LIN {X 0.072,Y -139.487,Z 751.117,A 0.000,B 0.000,C 90.000,E1 200.972} C_DIS
LIN {X 0.061,Y -138.989,Z 751.101,A 0.000,B 0.000,C 90.000,E1 198.181} C_DIS
LIN {X 0.022,Y -138.335,Z 751.054,A 0.000,B 0.000,C 90.000,E1 189.792} C_DIS
LIN {X 0.046,Y -139.420,Z 751.008,A 0.000,B 0.000,C 90.000,E1 181.375} C_DIS
LIN {X -0.041,Y -141.340,Z 750.972,A 0.000,B 0.000,C 90.000,E1 174.894} C_DIS
LIN {X 0.078,Y -142.696,Z 750.956,A 0.000,B 0.000,C 90.000,E1 172.064} C_DIS
LIN {X 0.038,Y -145.062,Z 750.930,A 0.000,B 0.000,C 90.000,E1 167.465} C_DIS
LIN {X 0.034,Y -147.687,Z 750.910,A 0.000,B 0.000,C 90.000,E1 163.795} C_DIS
LIN {X -0.074,Y -150.334,Z 750.890,A 0.000,B 0.000,C 90.000,E1 160.188} C_DIS
LIN {X -0.003,Y -153.753,Z 750.870,A 0.000,B 0.000,C 90.000,E1 156.538} C_DIS
LIN {X -0.012,Y -157.166,Z 750.850,A 0.000,B 0.000,C 90.000,E1 152.948} C_DIS
LIN {X -0.078,Y -161.320,Z 750.830,A 0.000,B 0.000,C 90.000,E1 149.410} C_DIS
LIN {X 0.075,Y -164.434,Z 750.815,A 0.000,B 0.000,C 90.000,E1 146.707} C_DIS
LIN {X 0.070,Y -169.120,Z 750.796,A 0.000,B 0.000,C 90.000,E1 143.210} C_DIS
LIN {X 0.018,Y -171.673,Z 750.786,A 0.000,B 0.000,C 90.000,E1 141.492} C_DIS
LIN {X -0.070,Y -176.641,Z 750.767,A 0.000,B 0.000,C 90.000,E1 138.081} C_DIS
LIN {X 0.057,Y -180.939,Z 750.753,A 0.000,B 0.000,C 90.000,E1 135.486} C_DIS
LIN {X 0.045,Y -186.359,Z 750.734,A 0.000,B 0.000,C 90.000,E1 132.123} C_DIS
LIN {X 0.004,Y -191.446,Z 750.719,A 0.000,B 0.000,C 90.000,E1 129.358} C_DIS
LIN {X 0.019,Y -192.042,Z 750.717,A 0.000,B 0.000,C 90.000,E1 128.991} C_DIS
LIN {X -0.007,Y -291.468,Z 750.717,A 0.000,B 0.000,C 90.000,E1 128.991} C_DIS
LIN {X -0.087,Y -296.497,Z 750.716,A 0.000,B 0.000,C 90.000,E1 128.830} C_DIS
LIN {X 0.018,Y -299.370,Z 750.714,A 0.000,B 0.000,C 90.000,E1 128.588} C_DIS
LIN {X -0.036,Y -303.124,Z 750.712,A 0.000,B 0.000,C 90.000,E1 128.141} C_DIS
LIN {X -0.019,Y -304.997,Z 750.710,A 0.000,B 0.000,C 90.000,E1 127.810} C_DIS
LIN {X 0.187,Y -306.459,Z 750.708,A 0.000,B 0.000,C 90.000,E1 127.443} C_DIS
LIN {X 0.173,Y -308.546,Z 750.705,A 0.000,B 0.000,C 90.000,E1 126.790} C_DIS
LIN {X -0.011,Y -318.461,Z 750.687,A 0.000,B 0.000,C 90.000,E1 123.579} C_DIS
LIN {X -0.052,Y -328.690,Z 750.671,A 0.000,B 0.000,C 90.000,E1 120.718} C_DIS
LIN {X -0.027,Y -340.261,Z 750.655,A 0.000,B 0.000,C 90.000,E1 117.897} C_DIS
LIN {X -0.136,Y -353.272,Z 750.640,A 0.000,B 0.000,C 90.000,E1 115.155} C_DIS
LIN {X 0.090,Y -366.144,Z 750.626,A 0.000,B 0.000,C 90.000,E1 112.717} C_DIS
LIN {X 0.031,Y -380.339,Z 750.613,A 0.000,B 0.000,C 90.000,E1 110.375} C_DIS
LIN {X 0.187,Y -395.960,Z 750.600,A 0.000,B 0.000,C 90.000,E1 108.055} C_DIS
LIN {X -0.022,Y -413.120,Z 750.588,A 0.000,B 0.000,C 90.000,E1 105.843} C_DIS
LIN {X 0.073,Y -431.944,Z 750.576,A 0.000,B 0.000,C 90.000,E1 103.647} C_DIS
LIN {X 0.019,Y -451.968,Z 750.564,A 0.000,B 0.000,C 90.000,E1 101.591} C_DIS
LIN {X 0.143,Y -467.357,Z 750.556,A 0.000,B 0.000,C 90.000,E1 100.141} C_DIS
LIN {X 0.178,Y -469.582,Z 750.555,A 0.000,B 0.000,C 90.000,E1 99.905} C_DIS
LIN {X 0.030,Y -471.399,Z 750.554,A 0.000,B 0.000,C 90.000,E1 99.670} C_DIS
LIN {X -0.120,Y -472.764,Z 750.552,A 0.000,B 0.000,C 90.000,E1 99.434} C_DIS
LIN {X -0.015,Y -474.484,Z 750.549,A 0.000,B 0.000,C 90.000,E1 98.916} C_DIS
LIN {X 0.102,Y -475.129,Z 750.547,A 0.000,B 0.000,C 90.000,E1 98.398} C_DIS
LIN {X -0.240,Y -474.807,Z 750.544,A 0.000,B 0.000,C 90.000,E1 97.936} C_DIS
LIN {X -0.045,Y -473.473,Z 750.541,A 0.000,B 0.000,C 90.000,E1 97.409} C_DIS
LIN {X -0.245,Y -472.363,Z 750.540,A 0.000,B 0.000,C 90.000,E1 97.182} C_DIS
LIN {X 0.198,Y -467.575,Z 750.536,A 0.000,B 0.000,C 90.000,E1 96.372} C_DIS
LIN {X -0.019,Y -451.599,Z 750.521,A 0.000,B 0.000,C 90.000,E1 93.841} C_DIS
LIN {X -0.186,Y -439.674,Z 750.510,A 0.000,B 0.000,C 90.000,E1 91.776} C_DIS
LIN {X 0.206,Y -432.077,Z 750.502,A 0.000,B 0.000,C 90.000,E1 90.401} C_DIS
LIN {X -0.117,Y -421.060,Z 750.492,A 0.000,B 0.000,C 90.000,E1 88.568} C_DIS
LIN {X 0.197,Y -410.004,Z 750.481,A 0.000,B 0.000,C 90.000,E1 86.617} C_DIS
LIN {X -0.167,Y -400.346,Z 750.472,A 0.000,B 0.000,C 90.000,E1 85.008} C_DIS
LIN {X 0.186,Y -387.551,Z 750.460,A 0.000,B 0.000,C 90.000,E1 82.704} C_DIS
LIN {X -0.043,Y -373.543,Z 750.445,A 0.000,B 0.000,C 90.000,E1 80.151} C_DIS
LIN {X -0.102,Y -361.605,Z 750.432,A 0.000,B 0.000,C 90.000,E1 77.813} C_DIS
LIN {X -0.027,Y -350.077,Z 750.419,A 0.000,B 0.000,C 90.000,E1 75.408} C_DIS
LIN {X 0.024,Y -338.783,Z 750.405,A 0.000,B 0.000,C 90.000,E1 72.960} C_DIS
LIN {X -0.133,Y -326.444,Z 750.390,A 0.000,B 0.000,C 90.000,E1 70.188} C_DIS
LIN {X 0.059,Y -313.531,Z 750.372,A 0.000,B 0.000,C 90.000,E1 66.975} C_DIS
LIN {X 0.121,Y -300.774,Z 750.352,A 0.000,B 0.000,C 90.000,E1 63.384} C_DIS
LIN {X 0.056,Y -290.366,Z 750.334,A 0.000,B 0.000,C 90.000,E1 60.078} C_DIS
LIN {X 0.009,Y -280.599,Z 750.315,A 0.000,B 0.000,C 90.000,E1 56.707} C_DIS
LIN {X -0.136,Y -273.069,Z 750.300,A 0.000,B 0.000,C 90.000,E1 53.989} C_DIS
LIN {X 0.017,Y -265.664,Z 750.284,A 0.000,B 0.000,C 90.000,E1 51.170} C_DIS
LIN {X 0.004,Y -259.989,Z 750.273,A 0.000,B 0.000,C 90.000,E1 49.057} C_DIS
LIN {X 0.056,Y -254.309,Z 750.261,A 0.000,B 0.000,C 90.000,E1 46.905} C_DIS
LIN {X -0.012,Y -248.565,Z 750.249,A 0.000,B 0.000,C 90.000,E1 44.757} C_DIS
LIN {X 0.160,Y -242.844,Z 750.236,A 0.000,B 0.000,C 90.000,E1 42.528} C_DIS
LIN {X -0.147,Y -235.195,Z 750.220,A 0.000,B 0.000,C 90.000,E1 39.644} C_DIS
LIN {X 0.087,Y -227.868,Z 750.203,A 0.000,B 0.000,C 90.000,E1 36.583} C_DIS
LIN {X -0.051,Y -219.365,Z 750.182,A 0.000,B 0.000,C 90.000,E1 32.801} C_DIS
LIN {X 0.065,Y -213.121,Z 750.165,A 0.000,B 0.000,C 90.000,E1 29.667} C_DIS
LIN {X 0.003,Y -207.678,Z 750.147,A 0.000,B 0.000,C 90.000,E1 26.539} C_DIS
LIN {X -0.103,Y -201.882,Z 750.125,A 0.000,B 0.000,C 90.000,E1 22.589} C_DIS
LIN {X -0.047,Y -197.159,Z 750.103,A 0.000,B 0.000,C 90.000,E1 18.544} C_DIS
LIN {X -0.070,Y -193.575,Z 750.080,A 0.000,B 0.000,C 90.000,E1 14.481} C_DIS
LIN {X 0.078,Y -190.269,Z 750.048,A 0.000,B 0.000,C 90.000,E1 8.690} C_DIS
LIN {X -0.039,Y -191.325,Z 749.961,A 0.000,B 0.000,C 90.000,E1 352.932} C_DIS
LIN {X -0.014,Y -194.658,Z 749.933,A 0.000,B 0.000,C 90.000,E1 347.993} C_DIS
LIN {X -0.037,Y -198.529,Z 749.911,A 0.000,B 0.000,C 90.000,E1 343.921} C_DIS
LIN {X -0.043,Y -203.397,Z 749.888,A 0.000,B 0.000,C 90.000,E1 339.880} C_DIS
LIN {X 0.004,Y -209.211,Z 749.866,A 0.000,B 0.000,C 90.000,E1 335.869} C_DIS
LIN {X 0.101,Y -215.898,Z 749.844,A 0.000,B 0.000,C 90.000,E1 331.897} C_DIS
LIN {X -0.033,Y -223.327,Z 749.822,A 0.000,B 0.000,C 90.000,E1 328.043} C_DIS
LIN {X 0.046,Y -231.309,Z 749.801,A 0.000,B 0.000,C 90.000,E1 324.196} C_DIS
LIN {X 0.029,Y -239.935,Z 749.780,A 0.000,B 0.000,C 90.000,E1 320.436} C_DIS
LIN {X 0.035,Y -247.397,Z 749.764,A 0.000,B 0.000,C 90.000,E1 317.472} C_DIS
LIN {X 0.063,Y -256.588,Z 749.746,A 0.000,B 0.000,C 90.000,E1 314.190} C_DIS
LIN {X 0.076,Y -267.646,Z 749.726,A 0.000,B 0.000,C 90.000,E1 310.620} C_DIS
LIN {X -0.048,Y -279.888,Z 749.706,A 0.000,B 0.000,C 90.000,E1 307.156} C_DIS
LIN {X 0.017,Y -291.945,Z 749.689,A 0.000,B 0.000,C 90.000,E1 304.072} C_DIS
LIN {X 0.091,Y -304.024,Z 749.674,A 0.000,B 0.000,C 90.000,E1 301.386} C_DIS
LIN {X -0.036,Y -320.894,Z 749.656,A 0.000,B 0.000,C 90.000,E1 298.153} C_DIS
LIN {X 0.011,Y -333.660,Z 749.644,A 0.000,B 0.000,C 90.000,E1 295.924} C_DIS
LIN {X 0.062,Y -351.261,Z 749.629,A 0.000,B 0.000,C 90.000,E1 293.131} C_DIS
LIN {X 0.151,Y -372.539,Z 749.612,A 0.000,B 0.000,C 90.000,E1 290.120} C_DIS
LIN {X 0.183,Y -393.526,Z 749.597,A 0.000,B 0.000,C 90.000,E1 287.511} C_DIS
LIN {X 0.041,Y -408.077,Z 749.588,A 0.000,B 0.000,C 90.000,E1 285.843} C_DIS
LIN {X 0.032,Y -422.254,Z 749.579,A 0.000,B 0.000,C 90.000,E1 284.189} C_DIS
LIN {X 0.099,Y -433.890,Z 749.571,A 0.000,B 0.000,C 90.000,E1 282.827} C_DIS
LIN {X -0.189,Y -445.013,Z 749.564,A 0.000,B 0.000,C 90.000,E1 281.535} C_DIS
LIN {X 0.029,Y -455.464,Z 749.557,A 0.000,B 0.000,C 90.000,E1 280.197} C_DIS
LIN {X -0.040,Y -465.472,Z 749.549,A 0.000,B 0.000,C 90.000,E1 278.916} C_DIS
LIN {X 0.174,Y -473.116,Z 749.544,A 0.000,B 0.000,C 90.000,E1 277.871} C_DIS
LIN {X 0.079,Y -478.362,Z 749.540,A 0.000,B 0.000,C 90.000,E1 277.125} C_DIS
LIN {X 0.095,Y -482.916,Z 749.535,A 0.000,B 0.000,C 90.000,E1 276.372} C_DIS
LIN {X 0.091,Y -486.699,Z 749.531,A 0.000,B 0.000,C 90.000,E1 275.625} C_DIS
LIN {X -0.198,Y -488.806,Z 749.529,A 0.000,B 0.000,C 90.000,E1 275.163} C_DIS
LIN {X 0.010,Y -490.520,Z 749.526,A 0.000,B 0.000,C 90.000,E1 274.645} C_DIS
LIN {X 0.187,Y -491.850,Z 749.523,A 0.000,B 0.000,C 90.000,E1 274.131} C_DIS
LIN {X -0.079,Y -492.733,Z 749.520,A 0.000,B 0.000,C 90.000,E1 273.669} C_DIS
LIN {X 0.121,Y -493.241,Z 749.518,A 0.000,B 0.000,C 90.000,E1 273.154} C_DIS
LIN {X -0.139,Y -493.319,Z 749.515,A 0.000,B 0.000,C 90.000,E1 272.694} C_DIS
LIN {X 0.074,Y -492.950,Z 749.512,A 0.000,B 0.000,C 90.000,E1 272.178} C_DIS
LIN {X -0.189,Y -492.180,Z 749.509,A 0.000,B 0.000,C 90.000,E1 271.718} C_DIS
LIN {X 0.022,Y -490.939,Z 749.507,A 0.000,B 0.000,C 90.000,E1 271.203} C_DIS
LIN {X 0.229,Y -489.215,Z 749.504,A 0.000,B 0.000,C 90.000,E1 270.688} C_DIS
LIN {X -0.060,Y -486.892,Z 749.501,A 0.000,B 0.000,C 90.000,E1 270.229} C_DIS
LIN {X 0.124,Y -483.960,Z 749.498,A 0.000,B 0.000,C 90.000,E1 269.714} C_DIS
LIN {X -0.191,Y -480.212,Z 749.496,A 0.000,B 0.000,C 90.000,E1 269.255} C_DIS
LIN {X 0.123,Y -478.066,Z 749.494,A 0.000,B 0.000,C 90.000,E1 268.969} C_DIS
LIN {X -0.196,Y -472.976,Z 749.492,A 0.000,B 0.000,C 90.000,E1 268.511} C_DIS
LIN {X 0.214,Y -467.101,Z 749.489,A 0.000,B 0.000,C 90.000,E1 267.993} C_DIS
LIN {X -0.175,Y -463.848,Z 749.488,A 0.000,B 0.000,C 90.000,E1 267.822} C_DIS
LIN {X 0.003,Y -457.103,Z 749.486,A 0.000,B 0.000,C 90.000,E1 267.421} C_DIS
LIN {X -0.218,Y -449.917,Z 749.484,A 0.000,B 0.000,C 90.000,E1 267.135} C_DIS
LIN {X 0.091,Y -442.331,Z 749.483,A 0.000,B 0.000,C 90.000,E1 266.846} C_DIS
LIN {X -0.040,Y -434.176,Z 749.482,A 0.000,B 0.000,C 90.000,E1 266.674} C_DIS
LIN {X -0.107,Y -429.962,Z 749.481,A 0.000,B 0.000,C 90.000,E1 266.617} C_DIS
LIN {X -0.170,Y -423.466,Z 749.481,A 0.000,B 0.000,C 90.000,E1 266.560} C_DIS
LIN {X 0.108,Y -419.173,Z 749.481,A 0.000,B 0.000,C 90.000,E1 266.502} C_DIS
LIN {X 0.016,Y -180.949,Z 749.481,A 0.000,B 0.000,C 90.000,E1 266.502} C_DIS
LIN {X -0.020,Y -180.796,Z 749.471,A 0.000,B 0.000,C 90.000,E1 264.780} C_DIS
LIN {X 0.054,Y -178.895,Z 749.443,A 0.000,B 0.000,C 90.000,E1 259.690} C_DIS
LIN {X -0.041,Y -175.938,Z 749.415,A 0.000,B 0.000,C 90.000,E1 254.629} C_DIS
LIN {X 0.075,Y -175.389,Z 749.410,A 0.000,B 0.000,C 90.000,E1 253.740} C_DIS
LIN {X -0.090,Y -172.160,Z 749.386,A 0.000,B 0.000,C 90.000,E1 249.518} C_DIS
LIN {X -0.051,Y -171.627,Z 749.381,A 0.000,B 0.000,C 90.000,E1 248.646} C_DIS
LIN {X -0.055,Y -167.850,Z 749.357,A 0.000,B 0.000,C 90.000,E1 244.332} C_DIS
LIN {X 0.036,Y -166.581,Z 749.348,A 0.000,B 0.000,C 90.000,E1 242.564} C_DIS
LIN {X 0.022,Y -162.572,Z 749.323,A 0.000,B 0.000,C 90.000,E1 238.201} C_DIS
LIN {X 0.082,Y -161.253,Z 749.314,A 0.000,B 0.000,C 90.000,E1 236.421} C_DIS
LIN {X -0.008,Y -157.256,Z 749.289,A 0.000,B 0.000,C 90.000,E1 232.029} C_DIS
LIN {X 0.039,Y -155.978,Z 749.279,A 0.000,B 0.000,C 90.000,E1 230.231} C_DIS
LIN {X 0.095,Y -152.233,Z 749.254,A 0.000,B 0.000,C 90.000,E1 225.729} C_DIS
LIN {X 0.005,Y -150.475,Z 749.239,A 0.000,B 0.000,C 90.000,E1 223.056} C_DIS
LIN {X -0.066,Y -147.200,Z 749.214,A 0.000,B 0.000,C 90.000,E1 218.543} C_DIS
LIN {X -0.012,Y -145.219,Z 749.194,A 0.000,B 0.000,C 90.000,E1 214.865} C_DIS
LIN {X 0.016,Y -142.349,Z 749.163,A 0.000,B 0.000,C 90.000,E1 209.333} C_DIS
LIN {X -0.057,Y -141.736,Z 749.153,A 0.000,B 0.000,C 90.000,E1 207.513} C_DIS
LIN {X 0.051,Y -139.485,Z 749.117,A 0.000,B 0.000,C 90.000,E1 200.972} C_DIS
LIN {X 0.040,Y -138.986,Z 749.101,A 0.000,B 0.000,C 90.000,E1 198.181} C_DIS
LIN {X 0.001,Y -138.335,Z 749.054,A 0.000,B 0.000,C 90.000,E1 189.792} C_DIS
LIN {X 0.025,Y -139.423,Z 749.008,A 0.000,B 0.000,C 90.000,E1 181.375} C_DIS
LIN {X -0.062,Y -141.343,Z 748.971,A 0.000,B 0.000,C 90.000,E1 174.894} C_DIS
LIN {X 0.055,Y -142.699,Z 748.956,A 0.000,B 0.000,C 90.000,E1 172.064} C_DIS
LIN {X 0.015,Y -145.068,Z 748.930,A 0.000,B 0.000,C 90.000,E1 167.465} C_DIS
LIN {X 0.011,Y -147.693,Z 748.910,A 0.000,B 0.000,C 90.000,E1 163.795} C_DIS
LIN {X 0.044,Y -150.342,Z 748.890,A 0.000,B 0.000,C 90.000,E1 160.134} C_DIS
LIN {X 0.039,Y -154.595,Z 748.865,A 0.000,B 0.000,C 90.000,E1 155.613} C_DIS
LIN {X 0.046,Y -158.135,Z 748.845,A 0.000,B 0.000,C 90.000,E1 152.025} C_DIS
LIN {X 0.006,Y -162.422,Z 748.825,A 0.000,B 0.000,C 90.000,E1 148.486} C_DIS
LIN {X -0.012,Y -166.678,Z 748.805,A 0.000,B 0.000,C 90.000,E1 144.975} C_DIS
LIN {X -0.006,Y -171.684,Z 748.786,A 0.000,B 0.000,C 90.000,E1 141.492} C_DIS
LIN {X -0.096,Y -176.655,Z 748.767,A 0.000,B 0.000,C 90.000,E1 138.081} C_DIS
LIN {X 0.031,Y -180.951,Z 748.753,A 0.000,B 0.000,C 90.000,E1 135.486} C_DIS
LIN {X 0.019,Y -186.373,Z 748.734,A 0.000,B 0.000,C 90.000,E1 132.123} C_DIS
LIN {X -0.020,Y -191.458,Z 748.719,A 0.000,B 0.000,C 90.000,E1 129.358} C_DIS
LIN {X -0.058,Y -192.006,Z 748.717,A 0.000,B 0.000,C 90.000,E1 129.036} C_DIS
LIN {X 0.099,Y -291.247,Z 748.717,A 0.000,B 0.000,C 90.000,E1 128.991} C_DIS
LIN {X -0.128,Y -296.846,Z 748.716,A 0.000,B 0.000,C 90.000,E1 128.830} C_DIS
LIN {X -0.071,Y -299.665,Z 748.714,A 0.000,B 0.000,C 90.000,E1 128.588} C_DIS
LIN {X -0.016,Y -303.427,Z 748.712,A 0.000,B 0.000,C 90.000,E1 128.096} C_DIS
LIN {X 0.175,Y -305.229,Z 748.710,A 0.000,B 0.000,C 90.000,E1 127.729} C_DIS
LIN {X -0.063,Y -306.637,Z 748.708,A 0.000,B 0.000,C 90.000,E1 127.443} C_DIS
LIN {X -0.077,Y -308.656,Z 748.704,A 0.000,B 0.000,C 90.000,E1 126.790} C_DIS
LIN {X 0.175,Y -318.592,Z 748.686,A 0.000,B 0.000,C 90.000,E1 123.499} C_DIS
LIN {X -0.028,Y -328.841,Z 748.670,A 0.000,B 0.000,C 90.000,E1 120.669} C_DIS
LIN {X 0.010,Y -340.434,Z 748.655,A 0.000,B 0.000,C 90.000,E1 117.847} C_DIS
LIN {X 0.065,Y -353.469,Z 748.639,A 0.000,B 0.000,C 90.000,E1 115.079} C_DIS
LIN {X -0.041,Y -366.363,Z 748.626,A 0.000,B 0.000,C 90.000,E1 112.695} C_DIS
LIN {X -0.115,Y -380.583,Z 748.613,A 0.000,B 0.000,C 90.000,E1 110.355} C_DIS
LIN {X -0.096,Y -396.231,Z 748.600,A 0.000,B 0.000,C 90.000,E1 108.055} C_DIS
LIN {X 0.086,Y -413.419,Z 748.588,A 0.000,B 0.000,C 90.000,E1 105.788} C_DIS
LIN {X 0.199,Y -432.274,Z 748.576,A 0.000,B 0.000,C 90.000,E1 103.592} C_DIS
LIN {X 0.176,Y -452.311,Z 748.564,A 0.000,B 0.000,C 90.000,E1 101.535} C_DIS
LIN {X -0.135,Y -467.700,Z 748.556,A 0.000,B 0.000,C 90.000,E1 100.141} C_DIS
LIN {X -0.098,Y -469.835,Z 748.555,A 0.000,B 0.000,C 90.000,E1 99.905} C_DIS
LIN {X 0.215,Y -471.594,Z 748.554,A 0.000,B 0.000,C 90.000,E1 99.613} C_DIS
LIN {X 0.062,Y -472.914,Z 748.552,A 0.000,B 0.000,C 90.000,E1 99.378} C_DIS
LIN {X 0.170,Y -474.562,Z 748.549,A 0.000,B 0.000,C 90.000,E1 98.859} C_DIS
LIN {X -0.182,Y -475.147,Z 748.547,A 0.000,B 0.000,C 90.000,E1 98.398} C_DIS
LIN {X 0.013,Y -474.766,Z 748.544,A 0.000,B 0.000,C 90.000,E1 97.871} C_DIS
LIN {X 0.143,Y -473.366,Z 748.541,A 0.000,B 0.000,C 90.000,E1 97.352} C_DIS
LIN {X -0.056,Y -472.214,Z 748.540,A 0.000,B 0.000,C 90.000,E1 97.125} C_DIS
LIN {X 0.014,Y -464.087,Z 748.533,A 0.000,B 0.000,C 90.000,E1 95.853} C_DIS
LIN {X -0.084,Y -449.918,Z 748.520,A 0.000,B 0.000,C 90.000,E1 93.555} C_DIS
LIN {X 0.153,Y -438.029,Z 748.508,A 0.000,B 0.000,C 90.000,E1 91.432} C_DIS
LIN {X -0.195,Y -428.810,Z 748.499,A 0.000,B 0.000,C 90.000,E1 89.885} C_DIS
LIN {X -0.039,Y -416.195,Z 748.487,A 0.000,B 0.000,C 90.000,E1 87.707} C_DIS
LIN {X 0.084,Y -406.663,Z 748.478,A 0.000,B 0.000,C 90.000,E1 86.045} C_DIS
LIN {X 0.187,Y -393.805,Z 748.466,A 0.000,B 0.000,C 90.000,E1 83.799} C_DIS
LIN {X 0.069,Y -379.611,Z 748.451,A 0.000,B 0.000,C 90.000,E1 81.254} C_DIS
LIN {X 0.067,Y -365.956,Z 748.437,A 0.000,B 0.000,C 90.000,E1 78.634} C_DIS
LIN {X -0.147,Y -352.883,Z 748.422,A 0.000,B 0.000,C 90.000,E1 75.992} C_DIS
LIN {X -0.109,Y -340.118,Z 748.407,A 0.000,B 0.000,C 90.000,E1 73.251} C_DIS
LIN {X 0.063,Y -326.403,Z 748.390,A 0.000,B 0.000,C 90.000,E1 70.115} C_DIS
LIN {X 0.061,Y -312.299,Z 748.370,A 0.000,B 0.000,C 90.000,E1 66.613} C_DIS
LIN {X -0.086,Y -300.847,Z 748.352,A 0.000,B 0.000,C 90.000,E1 63.384} C_DIS
LIN {X 0.005,Y -290.501,Z 748.334,A 0.000,B 0.000,C 90.000,E1 60.049} C_DIS
LIN {X -0.113,Y -282.676,Z 748.319,A 0.000,B 0.000,C 90.000,E1 57.375} C_DIS
LIN {X 0.028,Y -275.151,Z 748.303,A 0.000,B 0.000,C 90.000,E1 54.609} C_DIS
LIN {X 0.071,Y -267.765,Z 748.288,A 0.000,B 0.000,C 90.000,E1 51.823} C_DIS
LIN {X -0.073,Y -262.158,Z 748.276,A 0.000,B 0.000,C 90.000,E1 49.747} C_DIS
LIN {X 0.021,Y -256.488,Z 748.264,A 0.000,B 0.000,C 90.000,E1 47.595} C_DIS
LIN {X 0.001,Y -250.772,Z 748.253,A 0.000,B 0.000,C 90.000,E1 45.445} C_DIS
LIN {X 0.029,Y -243.123,Z 748.236,A 0.000,B 0.000,C 90.000,E1 42.528} C_DIS
LIN {X 0.065,Y -235.458,Z 748.220,A 0.000,B 0.000,C 90.000,E1 39.564} C_DIS
LIN {X 0.063,Y -226.335,Z 748.199,A 0.000,B 0.000,C 90.000,E1 35.804} C_DIS
LIN {X -0.058,Y -217.967,Z 748.178,A 0.000,B 0.000,C 90.000,E1 32.005} C_DIS
LIN {X 0.026,Y -211.881,Z 748.160,A 0.000,B 0.000,C 90.000,E1 28.871} C_DIS
LIN {X 0.023,Y -206.610,Z 748.143,A 0.000,B 0.000,C 90.000,E1 25.720} C_DIS
LIN {X 0.070,Y -201.000,Z 748.121,A 0.000,B 0.000,C 90.000,E1 21.716} C_DIS
LIN {X 0.023,Y -196.516,Z 748.098,A 0.000,B 0.000,C 90.000,E1 17.692} C_DIS
LIN {X -0.079,Y -193.118,Z 748.076,A 0.000,B 0.000,C 90.000,E1 13.647} C_DIS
LIN {X 0.002,Y -190.076,Z 748.044,A 0.000,B 0.000,C 90.000,E1 7.871} C_DIS
LIN {X 0.013,Y -191.004,Z 747.965,A 0.000,B 0.000,C 90.000,E1 353.742} C_DIS
LIN {X -0.010,Y -194.082,Z 747.938,A 0.000,B 0.000,C 90.000,E1 348.814} C_DIS
LIN {X -0.099,Y -197.779,Z 747.915,A 0.000,B 0.000,C 90.000,E1 344.755} C_DIS
LIN {X -0.002,Y -202.419,Z 747.893,A 0.000,B 0.000,C 90.000,E1 340.678} C_DIS
LIN {X 0.016,Y -208.066,Z 747.870,A 0.000,B 0.000,C 90.000,E1 336.666} C_DIS
LIN {X -0.109,Y -214.576,Z 747.848,A 0.000,B 0.000,C 90.000,E1 332.743} C_DIS
LIN {X 0.010,Y -220.361,Z 747.831,A 0.000,B 0.000,C 90.000,E1 329.587} C_DIS
LIN {X 0.064,Y -228.120,Z 747.810,A 0.000,B 0.000,C 90.000,E1 325.722} C_DIS
LIN {X -0.002,Y -236.456,Z 747.789,A 0.000,B 0.000,C 90.000,E1 321.949} C_DIS
LIN {X -0.079,Y -245.497,Z 747.768,A 0.000,B 0.000,C 90.000,E1 318.243} C_DIS
LIN {X 0.067,Y -254.503,Z 747.750,A 0.000,B 0.000,C 90.000,E1 314.919} C_DIS
LIN {X -0.005,Y -265.379,Z 747.730,A 0.000,B 0.000,C 90.000,E1 311.353} C_DIS
LIN {X 0.079,Y -276.112,Z 747.712,A 0.000,B 0.000,C 90.000,E1 308.177} C_DIS
LIN {X 0.107,Y -289.157,Z 747.693,A 0.000,B 0.000,C 90.000,E1 304.739} C_DIS
LIN {X -0.054,Y -300.897,Z 747.678,A 0.000,B 0.000,C 90.000,E1 302.084} C_DIS
LIN {X -0.024,Y -315.630,Z 747.662,A 0.000,B 0.000,C 90.000,E1 299.127} C_DIS
LIN {X 0.095,Y -331.779,Z 747.646,A 0.000,B 0.000,C 90.000,E1 296.232} C_DIS
LIN {X -0.026,Y -351.201,Z 747.629,A 0.000,B 0.000,C 90.000,E1 293.153} C_DIS
LIN {X 0.201,Y -372.429,Z 747.612,A 0.000,B 0.000,C 90.000,E1 290.120} C_DIS
LIN {X 0.092,Y -393.397,Z 747.597,A 0.000,B 0.000,C 90.000,E1 287.528} C_DIS
LIN {X 0.045,Y -407.920,Z 747.588,A 0.000,B 0.000,C 90.000,E1 285.843} C_DIS
LIN {X -0.104,Y -419.752,Z 747.580,A 0.000,B 0.000,C 90.000,E1 284.481} C_DIS
LIN {X -0.074,Y -431.405,Z 747.573,A 0.000,B 0.000,C 90.000,E1 283.119} C_DIS
LIN {X 0.025,Y -442.630,Z 747.565,A 0.000,B 0.000,C 90.000,E1 281.771} C_DIS
LIN {X 0.053,Y -451.138,Z 747.560,A 0.000,B 0.000,C 90.000,E1 280.715} C_DIS
LIN {X -0.082,Y -461.283,Z 747.552,A 0.000,B 0.000,C 90.000,E1 279.434} C_DIS
LIN {X -0.152,Y -471.093,Z 747.545,A 0.000,B 0.000,C 90.000,E1 278.163} C_DIS
LIN {X -0.202,Y -476.548,Z 747.541,A 0.000,B 0.000,C 90.000,E1 277.409} C_DIS
LIN {X 0.210,Y -481.337,Z 747.537,A 0.000,B 0.000,C 90.000,E1 276.606} C_DIS
LIN {X 0.250,Y -485.402,Z 747.533,A 0.000,B 0.000,C 90.000,E1 275.853} C_DIS
LIN {X -0.215,Y -488.686,Z 747.529,A 0.000,B 0.000,C 90.000,E1 275.163} C_DIS
LIN {X -0.008,Y -490.411,Z 747.526,A 0.000,B 0.000,C 90.000,E1 274.645} C_DIS
LIN {X 0.169,Y -491.755,Z 747.523,A 0.000,B 0.000,C 90.000,E1 274.131} C_DIS
LIN {X -0.099,Y -492.645,Z 747.520,A 0.000,B 0.000,C 90.000,E1 273.669} C_DIS
LIN {X 0.102,Y -493.136,Z 747.518,A 0.000,B 0.000,C 90.000,E1 273.154} C_DIS
LIN {X -0.159,Y -493.214,Z 747.515,A 0.000,B 0.000,C 90.000,E1 272.694} C_DIS
LIN {X 0.052,Y -492.883,Z 747.512,A 0.000,B 0.000,C 90.000,E1 272.178} C_DIS
LIN {X -0.211,Y -492.103,Z 747.509,A 0.000,B 0.000,C 90.000,E1 271.718} C_DIS
LIN {X 0.000,Y -490.878,Z 747.507,A 0.000,B 0.000,C 90.000,E1 271.203} C_DIS
LIN {X 0.207,Y -489.152,Z 747.504,A 0.000,B 0.000,C 90.000,E1 270.688} C_DIS
LIN {X -0.083,Y -486.898,Z 747.501,A 0.000,B 0.000,C 90.000,E1 270.229} C_DIS
LIN {X 0.101,Y -484.007,Z 747.498,A 0.000,B 0.000,C 90.000,E1 269.714} C_DIS
LIN {X -0.213,Y -480.283,Z 747.496,A 0.000,B 0.000,C 90.000,E1 269.255} C_DIS
LIN {X 0.100,Y -478.149,Z 747.494,A 0.000,B 0.000,C 90.000,E1 268.969} C_DIS
LIN {X -0.214,Y -473.120,Z 747.492,A 0.000,B 0.000,C 90.000,E1 268.511} C_DIS
LIN {X 0.221,Y -467.280,Z 747.489,A 0.000,B 0.000,C 90.000,E1 267.993} C_DIS
LIN {X 0.176,Y -460.939,Z 747.487,A 0.000,B 0.000,C 90.000,E1 267.593} C_DIS
LIN {X 0.146,Y -454.087,Z 747.485,A 0.000,B 0.000,C 90.000,E1 267.249} C_DIS
LIN {X 0.170,Y -446.760,Z 747.483,A 0.000,B 0.000,C 90.000,E1 266.963} C_DIS
LIN {X -0.208,Y -439.116,Z 747.482,A 0.000,B 0.000,C 90.000,E1 266.788} C_DIS
LIN {X -0.162,Y -430.250,Z 747.481,A 0.000,B 0.000,C 90.000,E1 266.617} C_DIS
LIN {X 0.188,Y -423.557,Z 747.481,A 0.000,B 0.000,C 90.000,E1 266.502} C_DIS
LIN {X 0.059,Y -420.149,Z 747.481,A 0.000,B 0.000,C 90.000,E1 266.502} C_DIS
LIN {X -0.003,Y -180.948,Z 747.481,A 0.000,B 0.000,C 90.000,E1 266.502} C_DIS
LIN {X -0.023,Y -180.795,Z 747.471,A 0.000,B 0.000,C 90.000,E1 264.780} C_DIS
LIN {X 0.050,Y -178.894,Z 747.443,A 0.000,B 0.000,C 90.000,E1 259.690} C_DIS
LIN {X -0.044,Y -175.937,Z 747.415,A 0.000,B 0.000,C 90.000,E1 254.629} C_DIS
LIN {X 0.070,Y -175.388,Z 747.410,A 0.000,B 0.000,C 90.000,E1 253.740} C_DIS
LIN {X -0.093,Y -172.159,Z 747.386,A 0.000,B 0.000,C 90.000,E1 249.518} C_DIS
LIN {X -0.054,Y -171.627,Z 747.381,A 0.000,B 0.000,C 90.000,E1 248.646} C_DIS
LIN {X -0.058,Y -167.850,Z 747.357,A 0.000,B 0.000,C 90.000,E1 244.332} C_DIS
LIN {X 0.033,Y -166.579,Z 747.348,A 0.000,B 0.000,C 90.000,E1 242.564} C_DIS
LIN {X 0.019,Y -162.571,Z 747.323,A 0.000,B 0.000,C 90.000,E1 238.201} C_DIS
LIN {X 0.078,Y -161.253,Z 747.314,A 0.000,B 0.000,C 90.000,E1 236.421} C_DIS
LIN {X -0.012,Y -157.255,Z 747.289,A 0.000,B 0.000,C 90.000,E1 232.029} C_DIS
LIN {X 0.035,Y -155.977,Z 747.279,A 0.000,B 0.000,C 90.000,E1 230.231} C_DIS
LIN {X 0.092,Y -152.232,Z 747.254,A 0.000,B 0.000,C 90.000,E1 225.729} C_DIS
LIN {X 0.003,Y -150.474,Z 747.239,A 0.000,B 0.000,C 90.000,E1 223.056} C_DIS
LIN {X -0.069,Y -147.199,Z 747.214,A 0.000,B 0.000,C 90.000,E1 218.543} C_DIS
LIN {X -0.016,Y -145.218,Z 747.194,A 0.000,B 0.000,C 90.000,E1 214.865} C_DIS
LIN {X 0.013,Y -142.348,Z 747.163,A 0.000,B 0.000,C 90.000,E1 209.333} C_DIS
LIN {X -0.060,Y -141.736,Z 747.153,A 0.000,B 0.000,C 90.000,E1 207.513} C_DIS
LIN {X 0.048,Y -139.485,Z 747.117,A 0.000,B 0.000,C 90.000,E1 200.972} C_DIS
LIN {X 0.037,Y -138.986,Z 747.101,A 0.000,B 0.000,C 90.000,E1 198.181} C_DIS
LIN {X -0.002,Y -138.334,Z 747.054,A 0.000,B 0.000,C 90.000,E1 189.792} C_DIS
LIN {X 0.022,Y -139.423,Z 747.008,A 0.000,B 0.000,C 90.000,E1 181.375} C_DIS
LIN {X -0.065,Y -141.345,Z 746.971,A 0.000,B 0.000,C 90.000,E1 174.894} C_DIS
LIN {X 0.052,Y -142.699,Z 746.956,A 0.000,B 0.000,C 90.000,E1 172.064} C_DIS
LIN {X 0.012,Y -145.068,Z 746.930,A 0.000,B 0.000,C 90.000,E1 167.465} C_DIS
LIN {X 0.008,Y -147.693,Z 746.910,A 0.000,B 0.000,C 90.000,E1 163.795} C_DIS
LIN {X 0.041,Y -150.343,Z 746.890,A 0.000,B 0.000,C 90.000,E1 160.134} C_DIS
LIN {X 0.035,Y -154.597,Z 746.865,A 0.000,B 0.000,C 90.000,E1 155.613} C_DIS
LIN {X 0.042,Y -158.137,Z 746.845,A 0.000,B 0.000,C 90.000,E1 152.025} C_DIS
LIN {X 0.002,Y -162.423,Z 746.825,A 0.000,B 0.000,C 90.000,E1 148.486} C_DIS
LIN {X -0.016,Y -166.680,Z 746.805,A 0.000,B 0.000,C 90.000,E1 144.975} C_DIS
LIN {X 0.097,Y -171.686,Z 746.786,A 0.000,B 0.000,C 90.000,E1 141.457} C_DIS
LIN {X -0.100,Y -176.657,Z 746.767,A 0.000,B 0.000,C 90.000,E1 138.081} C_DIS
LIN {X 0.028,Y -180.953,Z 746.753,A 0.000,B 0.000,C 90.000,E1 135.486} C_DIS
LIN {X 0.015,Y -186.376,Z 746.734,A 0.000,B 0.000,C 90.000,E1 132.123} C_DIS
LIN {X -0.023,Y -191.460,Z 746.719,A 0.000,B 0.000,C 90.000,E1 129.358} C_DIS
LIN {X 0.020,Y -191.967,Z 746.717,A 0.000,B 0.000,C 90.000,E1 129.036} C_DIS
LIN {X -0.009,Y -291.155,Z 746.717,A 0.000,B 0.000,C 90.000,E1 129.036} C_DIS
LIN {X 0.098,Y -292.615,Z 746.717,A 0.000,B 0.000,C 90.000,E1 128.991} C_DIS
LIN {X -0.133,Y -297.119,Z 746.716,A 0.000,B 0.000,C 90.000,E1 128.830} C_DIS
LIN {X -0.129,Y -300.333,Z 746.714,A 0.000,B 0.000,C 90.000,E1 128.543} C_DIS
LIN {X -0.062,Y -304.004,Z 746.711,A 0.000,B 0.000,C 90.000,E1 128.016} C_DIS
LIN {X 0.130,Y -305.658,Z 746.709,A 0.000,B 0.000,C 90.000,E1 127.649} C_DIS
LIN {X -0.107,Y -306.956,Z 746.707,A 0.000,B 0.000,C 90.000,E1 127.363} C_DIS
LIN {X -0.047,Y -318.863,Z 746.686,A 0.000,B 0.000,C 90.000,E1 123.452} C_DIS
LIN {X -0.074,Y -329.151,Z 746.670,A 0.000,B 0.000,C 90.000,E1 120.590} C_DIS
LIN {X -0.034,Y -340.786,Z 746.654,A 0.000,B 0.000,C 90.000,E1 117.769} C_DIS
LIN {X -0.127,Y -353.867,Z 746.639,A 0.000,B 0.000,C 90.000,E1 115.027} C_DIS
LIN {X 0.113,Y -366.804,Z 746.626,A 0.000,B 0.000,C 90.000,E1 112.589} C_DIS
LIN {X 0.068,Y -381.071,Z 746.613,A 0.000,B 0.000,C 90.000,E1 110.248} C_DIS
LIN {X 0.119,Y -396.770,Z 746.600,A 0.000,B 0.000,C 90.000,E1 107.946} C_DIS
LIN {X 0.048,Y -414.013,Z 746.587,A 0.000,B 0.000,C 90.000,E1 105.717} C_DIS
LIN {X 0.064,Y -432.923,Z 746.575,A 0.000,B 0.000,C 90.000,E1 103.536} C_DIS
LIN {X 0.086,Y -452.980,Z 746.564,A 0.000,B 0.000,C 90.000,E1 101.478} C_DIS
LIN {X -0.110,Y -468.327,Z 746.556,A 0.000,B 0.000,C 90.000,E1 100.074} C_DIS
LIN {X -0.150,Y -470.304,Z 746.555,A 0.000,B 0.000,C 90.000,E1 99.849} C_DIS
LIN {X 0.165,Y -471.948,Z 746.553,A 0.000,B 0.000,C 90.000,E1 99.557} C_DIS
LIN {X 0.015,Y -473.181,Z 746.552,A 0.000,B 0.000,C 90.000,E1 99.321} C_DIS
LIN {X 0.125,Y -474.696,Z 746.549,A 0.000,B 0.000,C 90.000,E1 98.803} C_DIS
LIN {X -0.225,Y -475.167,Z 746.546,A 0.000,B 0.000,C 90.000,E1 98.341} C_DIS
LIN {X -0.030,Y -474.676,Z 746.543,A 0.000,B 0.000,C 90.000,E1 97.814} C_DIS
LIN {X 0.102,Y -473.148,Z 746.541,A 0.000,B 0.000,C 90.000,E1 97.296} C_DIS
LIN {X -0.098,Y -471.915,Z 746.539,A 0.000,B 0.000,C 90.000,E1 97.068} C_DIS
LIN {X -0.179,Y -458.844,Z 746.528,A 0.000,B 0.000,C 90.000,E1 95.049} C_DIS
LIN {X -0.075,Y -439.204,Z 746.509,A 0.000,B 0.000,C 90.000,E1 91.661} C_DIS
LIN {X 0.031,Y -430.046,Z 746.500,A 0.000,B 0.000,C 90.000,E1 90.057} C_DIS
LIN {X 0.099,Y -419.009,Z 746.490,A 0.000,B 0.000,C 90.000,E1 88.165} C_DIS
LIN {X -0.133,Y -409.552,Z 746.481,A 0.000,B 0.000,C 90.000,E1 86.560} C_DIS
LIN {X -0.057,Y -398.302,Z 746.470,A 0.000,B 0.000,C 90.000,E1 84.609} C_DIS
LIN {X -0.100,Y -385.581,Z 746.457,A 0.000,B 0.000,C 90.000,E1 82.356} C_DIS
LIN {X -0.005,Y -371.671,Z 746.443,A 0.000,B 0.000,C 90.000,E1 79.746} C_DIS
LIN {X -0.147,Y -358.385,Z 746.428,A 0.000,B 0.000,C 90.000,E1 77.117} C_DIS
LIN {X -0.003,Y -348.362,Z 746.417,A 0.000,B 0.000,C 90.000,E1 74.991} C_DIS
LIN {X 0.008,Y -337.111,Z 746.403,A 0.000,B 0.000,C 90.000,E1 72.543} C_DIS
LIN {X -0.125,Y -323.554,Z 746.386,A 0.000,B 0.000,C 90.000,E1 69.444} C_DIS
LIN {X -0.094,Y -309.780,Z 746.366,A 0.000,B 0.000,C 90.000,E1 65.921} C_DIS
LIN {X 0.093,Y -298.681,Z 746.348,A 0.000,B 0.000,C 90.000,E1 62.615} C_DIS
LIN {X -0.137,Y -288.554,Z 746.329,A 0.000,B 0.000,C 90.000,E1 59.331} C_DIS
LIN {X -0.074,Y -278.973,Z 746.311,A 0.000,B 0.000,C 90.000,E1 55.928} C_DIS
LIN {X 0.128,Y -271.587,Z 746.295,A 0.000,B 0.000,C 90.000,E1 53.130} C_DIS
LIN {X -0.117,Y -266.071,Z 746.284,A 0.000,B 0.000,C 90.000,E1 51.090} C_DIS
LIN {X 0.077,Y -260.436,Z 746.272,A 0.000,B 0.000,C 90.000,E1 48.933} C_DIS
LIN {X -0.055,Y -254.778,Z 746.260,A 0.000,B 0.000,C 90.000,E1 46.824} C_DIS
LIN {X -0.097,Y -247.117,Z 746.244,A 0.000,B 0.000,C 90.000,E1 43.947} C_DIS
LIN {X -0.118,Y -241.372,Z 746.232,A 0.000,B 0.000,C 90.000,E1 41.757} C_DIS
LIN {X 0.057,Y -233.723,Z 746.215,A 0.000,B 0.000,C 90.000,E1 38.749} C_DIS
LIN {X 0.050,Y -224.731,Z 746.194,A 0.000,B 0.000,C 90.000,E1 34.978} C_DIS
LIN {X 0.066,Y -216.491,Z 746.173,A 0.000,B 0.000,C 90.000,E1 31.131} C_DIS
LIN {X 0.004,Y -210.593,Z 746.156,A 0.000,B 0.000,C 90.000,E1 28.025} C_DIS
LIN {X 0.067,Y -205.510,Z 746.138,A 0.000,B 0.000,C 90.000,E1 24.847} C_DIS
LIN {X 0.026,Y -201.092,Z 746.120,A 0.000,B 0.000,C 90.000,E1 21.663} C_DIS
LIN {X -0.011,Y -196.609,Z 746.098,A 0.000,B 0.000,C 90.000,E1 17.638} C_DIS
LIN {X -0.101,Y -192.655,Z 746.071,A 0.000,B 0.000,C 90.000,E1 12.771} C_DIS
LIN {X -0.067,Y -189.917,Z 746.039,A 0.000,B 0.000,C 90.000,E1 7.004} C_DIS
LIN {X 0.018,Y -191.099,Z 745.965,A 0.000,B 0.000,C 90.000,E1 353.742} C_DIS
LIN {X -0.002,Y -194.182,Z 745.938,A 0.000,B 0.000,C 90.000,E1 348.814} C_DIS
LIN {X -0.088,Y -197.885,Z 745.915,A 0.000,B 0.000,C 90.000,E1 344.755} C_DIS
LIN {X 0.012,Y -202.516,Z 745.893,A 0.000,B 0.000,C 90.000,E1 340.678} C_DIS
LIN {X 0.034,Y -208.164,Z 745.870,A 0.000,B 0.000,C 90.000,E1 336.666} C_DIS
LIN {X -0.087,Y -214.684,Z 745.848,A 0.000,B 0.000,C 90.000,E1 332.743} C_DIS
LIN {X 0.003,Y -221.937,Z 745.827,A 0.000,B 0.000,C 90.000,E1 328.820} C_DIS
LIN {X 0.027,Y -229.804,Z 745.805,A 0.000,B 0.000,C 90.000,E1 324.975} C_DIS
LIN {X 0.149,Y -238.221,Z 745.784,A 0.000,B 0.000,C 90.000,E1 321.170} C_DIS
LIN {X 0.102,Y -247.471,Z 745.764,A 0.000,B 0.000,C 90.000,E1 317.472} C_DIS
LIN {X 0.134,Y -256.634,Z 745.746,A 0.000,B 0.000,C 90.000,E1 314.190} C_DIS
LIN {X 0.153,Y -267.690,Z 745.726,A 0.000,B 0.000,C 90.000,E1 310.620} C_DIS
LIN {X 0.032,Y -279.925,Z 745.706,A 0.000,B 0.000,C 90.000,E1 307.156} C_DIS
LIN {X 0.125,Y -290.598,Z 745.691,A 0.000,B 0.000,C 90.000,E1 304.405} C_DIS
LIN {X 0.006,Y -302.478,Z 745.676,A 0.000,B 0.000,C 90.000,E1 301.750} C_DIS
LIN {X -0.007,Y -319.078,Z 745.658,A 0.000,B 0.000,C 90.000,E1 298.487} C_DIS
LIN {X 0.109,Y -333.601,Z 745.644,A 0.000,B 0.000,C 90.000,E1 295.924} C_DIS
LIN {X 0.192,Y -353.199,Z 745.627,A 0.000,B 0.000,C 90.000,E1 292.823} C_DIS
LIN {X -0.096,Y -372.324,Z 745.612,A 0.000,B 0.000,C 90.000,E1 290.174} C_DIS
LIN {X 0.108,Y -390.872,Z 745.599,A 0.000,B 0.000,C 90.000,E1 287.819} C_DIS
LIN {X 0.010,Y -405.320,Z 745.590,A 0.000,B 0.000,C 90.000,E1 286.134} C_DIS
LIN {X -0.177,Y -417.207,Z 745.582,A 0.000,B 0.000,C 90.000,E1 284.773} C_DIS
LIN {X -0.027,Y -431.198,Z 745.573,A 0.000,B 0.000,C 90.000,E1 283.119} C_DIS
LIN {X 0.070,Y -442.400,Z 745.565,A 0.000,B 0.000,C 90.000,E1 281.771} C_DIS
LIN {X 0.096,Y -450.893,Z 745.560,A 0.000,B 0.000,C 90.000,E1 280.715} C_DIS
LIN {X -0.117,Y -461.022,Z 745.552,A 0.000,B 0.000,C 90.000,E1 279.443} C_DIS
LIN {X -0.115,Y -470.907,Z 745.545,A 0.000,B 0.000,C 90.000,E1 278.163} C_DIS
LIN {X -0.166,Y -476.340,Z 745.541,A 0.000,B 0.000,C 90.000,E1 277.409} C_DIS
LIN {X -0.234,Y -481.153,Z 745.537,A 0.000,B 0.000,C 90.000,E1 276.663} C_DIS
LIN {X -0.199,Y -485.231,Z 745.533,A 0.000,B 0.000,C 90.000,E1 275.910} C_DIS
LIN {X -0.183,Y -488.555,Z 745.529,A 0.000,B 0.000,C 90.000,E1 275.163} C_DIS
LIN {X 0.023,Y -490.281,Z 745.526,A 0.000,B 0.000,C 90.000,E1 274.645} C_DIS
LIN {X 0.199,Y -491.624,Z 745.523,A 0.000,B 0.000,C 90.000,E1 274.131} C_DIS
LIN {X -0.069,Y -492.525,Z 745.520,A 0.000,B 0.000,C 90.000,E1 273.669} C_DIS
LIN {X 0.130,Y -493.049,Z 745.518,A 0.000,B 0.000,C 90.000,E1 273.154} C_DIS
LIN {X -0.131,Y -493.124,Z 745.515,A 0.000,B 0.000,C 90.000,E1 272.694} C_DIS
LIN {X 0.080,Y -492.786,Z 745.512,A 0.000,B 0.000,C 90.000,E1 272.178} C_DIS
LIN {X -0.183,Y -492.028,Z 745.509,A 0.000,B 0.000,C 90.000,E1 271.718} C_DIS
LIN {X 0.026,Y -490.804,Z 745.507,A 0.000,B 0.000,C 90.000,E1 271.203} C_DIS
LIN {X 0.232,Y -489.125,Z 745.504,A 0.000,B 0.000,C 90.000,E1 270.688} C_DIS
LIN {X -0.057,Y -486.880,Z 745.501,A 0.000,B 0.000,C 90.000,E1 270.229} C_DIS
LIN {X 0.127,Y -484.031,Z 745.498,A 0.000,B 0.000,C 90.000,E1 269.714} C_DIS
LIN {X -0.188,Y -480.371,Z 745.496,A 0.000,B 0.000,C 90.000,E1 269.255} C_DIS
LIN {X -0.040,Y -475.833,Z 745.493,A 0.000,B 0.000,C 90.000,E1 268.740} C_DIS
LIN {X -0.215,Y -473.240,Z 745.492,A 0.000,B 0.000,C 90.000,E1 268.511} C_DIS
LIN {X 0.188,Y -467.344,Z 745.489,A 0.000,B 0.000,C 90.000,E1 267.993} C_DIS
LIN {X 0.123,Y -460.976,Z 745.487,A 0.000,B 0.000,C 90.000,E1 267.593} C_DIS
LIN {X 0.069,Y -454.084,Z 745.485,A 0.000,B 0.000,C 90.000,E1 267.249} C_DIS
LIN {X 0.083,Y -446.753,Z 745.483,A 0.000,B 0.000,C 90.000,E1 266.963} C_DIS
LIN {X 0.154,Y -439.149,Z 745.482,A 0.000,B 0.000,C 90.000,E1 266.731} C_DIS
LIN {X 0.203,Y -430.341,Z 745.481,A 0.000,B 0.000,C 90.000,E1 266.560} C_DIS
LIN {X -0.019,Y -420.049,Z 745.481,A 0.000,B 0.000,C 90.000,E1 266.502} C_DIS
LIN {X -0.039,Y -180.947,Z 745.481,A 0.000,B 0.000,C 90.000,E1 266.502} C_DIS
LIN {X -0.078,Y -180.789,Z 745.471,A 0.000,B 0.000,C 90.000,E1 264.780} C_DIS
LIN {X -0.003,Y -178.887,Z 745.443,A 0.000,B 0.000,C 90.000,E1 259.690} C_DIS
LIN {X 0.072,Y -175.930,Z 745.414,A 0.000,B 0.000,C 90.000,E1 254.574} C_DIS
LIN {X 0.018,Y -175.373,Z 745.410,A 0.000,B 0.000,C 90.000,E1 253.740} C_DIS
LIN {X 0.075,Y -172.148,Z 745.386,A 0.000,B 0.000,C 90.000,E1 249.444} C_DIS
LIN {X 0.053,Y -171.614,Z 745.381,A 0.000,B 0.000,C 90.000,E1 248.592} C_DIS
LIN {X 0.041,Y -167.836,Z 745.357,A 0.000,B 0.000,C 90.000,E1 244.280} C_DIS
LIN {X 0.058,Y -166.564,Z 745.348,A 0.000,B 0.000,C 90.000,E1 242.538} C_DIS
LIN {X -0.032,Y -162.557,Z 745.323,A 0.000,B 0.000,C 90.000,E1 238.201} C_DIS
LIN {X 0.028,Y -161.237,Z 745.313,A 0.000,B 0.000,C 90.000,E1 236.421} C_DIS
LIN {X 0.063,Y -157.241,Z 745.289,A 0.000,B 0.000,C 90.000,E1 231.984} C_DIS
LIN {X -0.015,Y -155.965,Z 745.279,A 0.000,B 0.000,C 90.000,E1 230.231} C_DIS
LIN {X 0.044,Y -152.219,Z 745.254,A 0.000,B 0.000,C 90.000,E1 225.729} C_DIS
LIN {X 0.064,Y -150.463,Z 745.239,A 0.000,B 0.000,C 90.000,E1 223.014} C_DIS
LIN {X 0.089,Y -147.188,Z 745.214,A 0.000,B 0.000,C 90.000,E1 218.463} C_DIS
LIN {X 0.056,Y -145.206,Z 745.194,A 0.000,B 0.000,C 90.000,E1 214.818} C_DIS
LIN {X -0.034,Y -142.341,Z 745.163,A 0.000,B 0.000,C 90.000,E1 209.333} C_DIS
LIN {X 0.020,Y -141.730,Z 745.153,A 0.000,B 0.000,C 90.000,E1 207.462} C_DIS
LIN {X 0.002,Y -139.481,Z 745.117,A 0.000,B 0.000,C 90.000,E1 200.972} C_DIS
LIN {X -0.010,Y -138.981,Z 745.101,A 0.000,B 0.000,C 90.000,E1 198.181} C_DIS
LIN {X -0.049,Y -138.333,Z 745.054,A 0.000,B 0.000,C 90.000,E1 189.792} C_DIS
LIN {X -0.024,Y -139.428,Z 745.008,A 0.000,B 0.000,C 90.000,E1 181.375} C_DIS
LIN {X 0.029,Y -141.353,Z 744.971,A 0.000,B 0.000,C 90.000,E1 174.837} C_DIS
LIN {X 0.006,Y -142.707,Z 744.956,A 0.000,B 0.000,C 90.000,E1 172.064} C_DIS
LIN {X -0.035,Y -145.080,Z 744.930,A 0.000,B 0.000,C 90.000,E1 167.465} C_DIS
LIN {X -0.039,Y -147.705,Z 744.910,A 0.000,B 0.000,C 90.000,E1 163.795} C_DIS
LIN {X 0.044,Y -150.358,Z 744.890,A 0.000,B 0.000,C 90.000,E1 160.115} C_DIS
LIN {X 0.063,Y -153.783,Z 744.870,A 0.000,B 0.000,C 90.000,E1 156.485} C_DIS
LIN {X -0.018,Y -157.195,Z 744.850,A 0.000,B 0.000,C 90.000,E1 152.922} C_DIS
LIN {X 0.065,Y -161.356,Z 744.830,A 0.000,B 0.000,C 90.000,E1 149.331} C_DIS
LIN {X 0.077,Y -165.559,Z 744.810,A 0.000,B 0.000,C 90.000,E1 145.801} C_DIS
LIN {X -0.040,Y -170.474,Z 744.791,A 0.000,B 0.000,C 90.000,E1 142.351} C_DIS
LIN {X 0.110,Y -175.356,Z 744.772,A 0.000,B 0.000,C 90.000,E1 138.852} C_DIS
LIN {X -0.027,Y -180.980,Z 744.753,A 0.000,B 0.000,C 90.000,E1 135.486} C_DIS
LIN {X -0.040,Y -186.405,Z 744.734,A 0.000,B 0.000,C 90.000,E1 132.123} C_DIS
LIN {X -0.077,Y -191.486,Z 744.719,A 0.000,B 0.000,C 90.000,E1 129.358} C_DIS
LIN {X -0.031,Y -191.934,Z 744.717,A 0.000,B 0.000,C 90.000,E1 129.072} C_DIS
LIN {X 0.090,Y -291.343,Z 744.717,A 0.000,B 0.000,C 90.000,E1 129.036} C_DIS
LIN {X -0.048,Y -292.792,Z 744.717,A 0.000,B 0.000,C 90.000,E1 129.036} C_DIS
LIN {X 0.011,Y -297.576,Z 744.715,A 0.000,B 0.000,C 90.000,E1 128.785} C_DIS
LIN {X 0.078,Y -300.809,Z 744.714,A 0.000,B 0.000,C 90.000,E1 128.463} C_DIS
LIN {X -0.029,Y -304.446,Z 744.711,A 0.000,B 0.000,C 90.000,E1 127.935} C_DIS
LIN {X -0.021,Y -305.985,Z 744.709,A 0.000,B 0.000,C 90.000,E1 127.604} C_DIS
LIN {X -0.070,Y -307.195,Z 744.707,A 0.000,B 0.000,C 90.000,E1 127.282} C_DIS
LIN {X -0.065,Y -318.009,Z 744.687,A 0.000,B 0.000,C 90.000,E1 123.706} C_DIS
LIN {X 0.154,Y -328.188,Z 744.671,A 0.000,B 0.000,C 90.000,E1 120.797} C_DIS
LIN {X -0.118,Y -339.700,Z 744.656,A 0.000,B 0.000,C 90.000,E1 118.025} C_DIS
LIN {X 0.218,Y -352.653,Z 744.640,A 0.000,B 0.000,C 90.000,E1 115.207} C_DIS
LIN {X 0.097,Y -365.467,Z 744.627,A 0.000,B 0.000,C 90.000,E1 112.823} C_DIS
LIN {X 0.010,Y -379.601,Z 744.614,A 0.000,B 0.000,C 90.000,E1 110.482} C_DIS
LIN {X 0.013,Y -395.154,Z 744.601,A 0.000,B 0.000,C 90.000,E1 108.181} C_DIS
LIN {X -0.106,Y -412.243,Z 744.589,A 0.000,B 0.000,C 90.000,E1 105.953} C_DIS
LIN {X -0.148,Y -430.989,Z 744.576,A 0.000,B 0.000,C 90.000,E1 103.772} C_DIS
LIN {X 0.171,Y -450.989,Z 744.565,A 0.000,B 0.000,C 90.000,E1 101.658} C_DIS
LIN {X -0.068,Y -468.794,Z 744.556,A 0.000,B 0.000,C 90.000,E1 100.018} C_DIS
LIN {X -0.103,Y -470.659,Z 744.554,A 0.000,B 0.000,C 90.000,E1 99.792} C_DIS
LIN {X 0.214,Y -472.219,Z 744.553,A 0.000,B 0.000,C 90.000,E1 99.500} C_DIS
LIN {X 0.065,Y -473.387,Z 744.552,A 0.000,B 0.000,C 90.000,E1 99.265} C_DIS
LIN {X 0.178,Y -474.797,Z 744.549,A 0.000,B 0.000,C 90.000,E1 98.746} C_DIS
LIN {X -0.101,Y -475.181,Z 744.546,A 0.000,B 0.000,C 90.000,E1 98.276} C_DIS
LIN {X 0.027,Y -474.601,Z 744.543,A 0.000,B 0.000,C 90.000,E1 97.757} C_DIS
LIN {X 0.158,Y -472.969,Z 744.540,A 0.000,B 0.000,C 90.000,E1 97.239} C_DIS
LIN {X 0.017,Y -471.669,Z 744.539,A 0.000,B 0.000,C 90.000,E1 97.004} C_DIS
LIN {X -0.061,Y -452.319,Z 744.522,A 0.000,B 0.000,C 90.000,E1 93.955} C_DIS
LIN {X -0.034,Y -438.955,Z 744.509,A 0.000,B 0.000,C 90.000,E1 91.604} C_DIS
LIN {X -0.087,Y -431.343,Z 744.502,A 0.000,B 0.000,C 90.000,E1 90.286} C_DIS
LIN {X 0.004,Y -420.336,Z 744.491,A 0.000,B 0.000,C 90.000,E1 88.396} C_DIS
LIN {X -0.111,Y -409.313,Z 744.480,A 0.000,B 0.000,C 90.000,E1 86.502} C_DIS
LIN {X -0.002,Y -398.085,Z 744.470,A 0.000,B 0.000,C 90.000,E1 84.546} C_DIS
LIN {X -0.091,Y -385.372,Z 744.457,A 0.000,B 0.000,C 90.000,E1 82.299} C_DIS
LIN {X 0.000,Y -369.998,Z 744.441,A 0.000,B 0.000,C 90.000,E1 79.398} C_DIS
LIN {X -0.155,Y -355.360,Z 744.425,A 0.000,B 0.000,C 90.000,E1 76.464} C_DIS
LIN {X -0.073,Y -345.359,Z 744.413,A 0.000,B 0.000,C 90.000,E1 74.338} C_DIS
LIN {X -0.032,Y -334.198,Z 744.399,A 0.000,B 0.000,C 90.000,E1 71.873} C_DIS
LIN {X 0.054,Y -320.857,Z 744.382,A 0.000,B 0.000,C 90.000,E1 68.720} C_DIS
LIN {X -0.006,Y -309.737,Z 744.366,A 0.000,B 0.000,C 90.000,E1 65.845} C_DIS
LIN {X 0.053,Y -298.718,Z 744.348,A 0.000,B 0.000,C 90.000,E1 62.564} C_DIS
LIN {X -0.035,Y -288.641,Z 744.329,A 0.000,B 0.000,C 90.000,E1 59.253} C_DIS
LIN {X -0.124,Y -279.128,Z 744.310,A 0.000,B 0.000,C 90.000,E1 55.881} C_DIS
LIN {X -0.142,Y -271.771,Z 744.295,A 0.000,B 0.000,C 90.000,E1 53.130} C_DIS
LIN {X -0.003,Y -266.275,Z 744.283,A 0.000,B 0.000,C 90.000,E1 51.009} C_DIS
LIN {X -0.174,Y -260.659,Z 744.272,A 0.000,B 0.000,C 90.000,E1 48.933} C_DIS
LIN {X 0.064,Y -254.995,Z 744.260,A 0.000,B 0.000,C 90.000,E1 46.743} C_DIS
LIN {X 0.008,Y -249.252,Z 744.248,A 0.000,B 0.000,C 90.000,E1 44.595} C_DIS
LIN {X 0.004,Y -241.578,Z 744.232,A 0.000,B 0.000,C 90.000,E1 41.676} C_DIS
LIN {X 0.032,Y -233.921,Z 744.215,A 0.000,B 0.000,C 90.000,E1 38.705} C_DIS
LIN {X -0.014,Y -224.917,Z 744.194,A 0.000,B 0.000,C 90.000,E1 34.945} C_DIS
LIN {X -0.115,Y -216.638,Z 744.173,A 0.000,B 0.000,C 90.000,E1 31.131} C_DIS
LIN {X 0.018,Y -210.736,Z 744.155,A 0.000,B 0.000,C 90.000,E1 27.975} C_DIS
LIN {X -0.007,Y -204.462,Z 744.133,A 0.000,B 0.000,C 90.000,E1 24.027} C_DIS
LIN {X 0.110,Y -200.221,Z 744.116,A 0.000,B 0.000,C 90.000,E1 20.791} C_DIS
LIN {X -0.086,Y -195.961,Z 744.093,A 0.000,B 0.000,C 90.000,E1 16.804} C_DIS
LIN {X -0.013,Y -192.246,Z 744.066,A 0.000,B 0.000,C 90.000,E1 11.883} C_DIS
LIN {X 0.048,Y -189.635,Z 744.029,A 0.000,B 0.000,C 90.000,E1 5.277} C_DIS
LIN {X 0.073,Y -190.829,Z 743.970,A 0.000,B 0.000,C 90.000,E1 354.552} C_DIS
LIN {X 0.005,Y -193.643,Z 743.942,A 0.000,B 0.000,C 90.000,E1 349.634} C_DIS
LIN {X 0.095,Y -197.176,Z 743.920,A 0.000,B 0.000,C 90.000,E1 345.519} C_DIS
LIN {X -0.067,Y -201.581,Z 743.897,A 0.000,B 0.000,C 90.000,E1 341.511} C_DIS
LIN {X -0.031,Y -207.075,Z 743.875,A 0.000,B 0.000,C 90.000,E1 337.486} C_DIS
LIN {X 0.001,Y -213.427,Z 743.853,A 0.000,B 0.000,C 90.000,E1 333.512} C_DIS
LIN {X -0.051,Y -220.533,Z 743.831,A 0.000,B 0.000,C 90.000,E1 329.616} C_DIS
LIN {X -0.009,Y -228.232,Z 743.810,A 0.000,B 0.000,C 90.000,E1 325.754} C_DIS
LIN {X -0.007,Y -234.844,Z 743.793,A 0.000,B 0.000,C 90.000,E1 322.718} C_DIS
LIN {X 0.015,Y -243.685,Z 743.772,A 0.000,B 0.000,C 90.000,E1 318.976} C_DIS
LIN {X -0.054,Y -253.494,Z 743.752,A 0.000,B 0.000,C 90.000,E1 315.324} C_DIS
LIN {X -0.160,Y -264.302,Z 743.732,A 0.000,B 0.000,C 90.000,E1 311.757} C_DIS
LIN {X 0.067,Y -274.887,Z 743.714,A 0.000,B 0.000,C 90.000,E1 308.543} C_DIS
LIN {X 0.059,Y -287.816,Z 743.695,A 0.000,B 0.000,C 90.000,E1 305.105} C_DIS
LIN {X 0.035,Y -300.949,Z 743.678,A 0.000,B 0.000,C 90.000,E1 302.084} C_DIS
LIN {X 0.015,Y -313.893,Z 743.664,A 0.000,B 0.000,C 90.000,E1 299.461} C_DIS
LIN {X -0.104,Y -331.722,Z 743.646,A 0.000,B 0.000,C 90.000,E1 296.283} C_DIS
LIN {X 0.075,Y -351.123,Z 743.629,A 0.000,B 0.000,C 90.000,E1 293.153} C_DIS
LIN {X -0.125,Y -369.993,Z 743.614,A 0.000,B 0.000,C 90.000,E1 290.482} C_DIS
LIN {X 0.160,Y -390.719,Z 743.599,A 0.000,B 0.000,C 90.000,E1 287.819} C_DIS
LIN {X 0.146,Y -407.519,Z 743.588,A 0.000,B 0.000,C 90.000,E1 285.843} C_DIS
LIN {X 0.014,Y -419.346,Z 743.580,A 0.000,B 0.000,C 90.000,E1 284.481} C_DIS
LIN {X 0.041,Y -430.974,Z 743.573,A 0.000,B 0.000,C 90.000,E1 283.119} C_DIS
LIN {X 0.136,Y -442.157,Z 743.565,A 0.000,B 0.000,C 90.000,E1 281.771} C_DIS
LIN {X 0.077,Y -450.625,Z 743.560,A 0.000,B 0.000,C 90.000,E1 280.725} C_DIS
LIN {X -0.055,Y -460.756,Z 743.552,A 0.000,B 0.000,C 90.000,E1 279.443} C_DIS
LIN {X -0.055,Y -470.667,Z 743.545,A 0.000,B 0.000,C 90.000,E1 278.163} C_DIS
LIN {X -0.107,Y -476.148,Z 743.541,A 0.000,B 0.000,C 90.000,E1 277.409} C_DIS
LIN {X -0.178,Y -480.979,Z 743.537,A 0.000,B 0.000,C 90.000,E1 276.663} C_DIS
LIN {X -0.144,Y -485.046,Z 743.533,A 0.000,B 0.000,C 90.000,E1 275.910} C_DIS
LIN {X -0.129,Y -488.376,Z 743.529,A 0.000,B 0.000,C 90.000,E1 275.163} C_DIS
LIN {X 0.076,Y -490.114,Z 743.526,A 0.000,B 0.000,C 90.000,E1 274.645} C_DIS
LIN {X -0.239,Y -491.459,Z 743.523,A 0.000,B 0.000,C 90.000,E1 274.188} C_DIS
LIN {X -0.017,Y -492.370,Z 743.520,A 0.000,B 0.000,C 90.000,E1 273.669} C_DIS
LIN {X 0.181,Y -492.878,Z 743.518,A 0.000,B 0.000,C 90.000,E1 273.154} C_DIS
LIN {X -0.080,Y -492.993,Z 743.515,A 0.000,B 0.000,C 90.000,E1 272.694} C_DIS
LIN {X 0.129,Y -492.682,Z 743.512,A 0.000,B 0.000,C 90.000,E1 272.178} C_DIS
LIN {X -0.134,Y -491.934,Z 743.509,A 0.000,B 0.000,C 90.000,E1 271.718} C_DIS
LIN {X 0.075,Y -490.746,Z 743.507,A 0.000,B 0.000,C 90.000,E1 271.203} C_DIS
LIN {X -0.210,Y -489.049,Z 743.504,A 0.000,B 0.000,C 90.000,E1 270.745} C_DIS
LIN {X -0.010,Y -486.875,Z 743.501,A 0.000,B 0.000,C 90.000,E1 270.229} C_DIS
LIN {X 0.178,Y -484.054,Z 743.499,A 0.000,B 0.000,C 90.000,E1 269.714} C_DIS
LIN {X -0.137,Y -480.456,Z 743.496,A 0.000,B 0.000,C 90.000,E1 269.255} C_DIS
LIN {X 0.011,Y -475.976,Z 743.493,A 0.000,B 0.000,C 90.000,E1 268.740} C_DIS
LIN {X -0.164,Y -473.346,Z 743.492,A 0.000,B 0.000,C 90.000,E1 268.511} C_DIS
LIN {X 0.207,Y -467.499,Z 743.489,A 0.000,B 0.000,C 90.000,E1 267.993} C_DIS
LIN {X 0.118,Y -461.171,Z 743.487,A 0.000,B 0.000,C 90.000,E1 267.593} C_DIS
LIN {X 0.076,Y -454.345,Z 743.485,A 0.000,B 0.000,C 90.000,E1 267.249} C_DIS
LIN {X 0.179,Y -450.570,Z 743.484,A 0.000,B 0.000,C 90.000,E1 267.078} C_DIS
LIN {X -0.001,Y -443.042,Z 743.482,A 0.000,B 0.000,C 90.000,E1 266.846} C_DIS
LIN {X 0.177,Y -434.326,Z 743.481,A 0.000,B 0.000,C 90.000,E1 266.617} C_DIS
LIN {X 0.107,Y -430.193,Z 743.481,A 0.000,B 0.000,C 90.000,E1 266.560} C_DIS
LIN {X -0.107,Y -420.036,Z 743.480,A 0.000,B 0.000,C 90.000,E1 266.502} C_DIS
LIN {X -0.077,Y -180.947,Z 743.480,A 0.000,B 0.000,C 90.000,E1 266.502} C_DIS
LIN {X 0.063,Y -180.785,Z 743.471,A 0.000,B 0.000,C 90.000,E1 264.723} C_DIS
LIN {X -0.042,Y -178.882,Z 743.443,A 0.000,B 0.000,C 90.000,E1 259.690} C_DIS
LIN {X 0.034,Y -175.924,Z 743.414,A 0.000,B 0.000,C 90.000,E1 254.574} C_DIS
LIN {X -0.021,Y -175.361,Z 743.410,A 0.000,B 0.000,C 90.000,E1 253.740} C_DIS
LIN {X 0.038,Y -172.141,Z 743.386,A 0.000,B 0.000,C 90.000,E1 249.444} C_DIS
LIN {X 0.015,Y -171.604,Z 743.381,A 0.000,B 0.000,C 90.000,E1 248.592} C_DIS
LIN {X 0.004,Y -167.827,Z 743.357,A 0.000,B 0.000,C 90.000,E1 244.280} C_DIS
LIN {X 0.021,Y -166.552,Z 743.347,A 0.000,B 0.000,C 90.000,E1 242.538} C_DIS
LIN {X -0.069,Y -162.547,Z 743.323,A 0.000,B 0.000,C 90.000,E1 238.201} C_DIS
LIN {X -0.009,Y -161.225,Z 743.313,A 0.000,B 0.000,C 90.000,E1 236.421} C_DIS
LIN {X 0.027,Y -157.231,Z 743.289,A 0.000,B 0.000,C 90.000,E1 231.984} C_DIS
LIN {X 0.050,Y -155.956,Z 743.279,A 0.000,B 0.000,C 90.000,E1 230.194} C_DIS
LIN {X 0.008,Y -152.209,Z 743.254,A 0.000,B 0.000,C 90.000,E1 225.729} C_DIS
LIN {X 0.030,Y -150.454,Z 743.239,A 0.000,B 0.000,C 90.000,E1 223.014} C_DIS
LIN {X 0.056,Y -147.180,Z 743.214,A 0.000,B 0.000,C 90.000,E1 218.463} C_DIS
LIN {X 0.023,Y -145.197,Z 743.193,A 0.000,B 0.000,C 90.000,E1 214.818} C_DIS
LIN {X 0.057,Y -142.336,Z 743.163,A 0.000,B 0.000,C 90.000,E1 209.283} C_DIS
LIN {X -0.014,Y -141.725,Z 743.153,A 0.000,B 0.000,C 90.000,E1 207.462} C_DIS
LIN {X -0.032,Y -139.479,Z 743.116,A 0.000,B 0.000,C 90.000,E1 200.972} C_DIS
LIN {X -0.042,Y -138.977,Z 743.101,A 0.000,B 0.000,C 90.000,E1 198.181} C_DIS
LIN {X 0.078,Y -138.331,Z 743.054,A 0.000,B 0.000,C 90.000,E1 189.726} C_DIS
LIN {X -0.057,Y -139.431,Z 743.008,A 0.000,B 0.000,C 90.000,E1 181.375} C_DIS
LIN {X 0.021,Y -140.956,Z 742.976,A 0.000,B 0.000,C 90.000,E1 175.755} C_DIS
LIN {X -0.028,Y -142.712,Z 742.956,A 0.000,B 0.000,C 90.000,E1 172.064} C_DIS
LIN {X 0.072,Y -145.088,Z 742.930,A 0.000,B 0.000,C 90.000,E1 167.409} C_DIS
LIN {X 0.068,Y -147.714,Z 742.910,A 0.000,B 0.000,C 90.000,E1 163.740} C_DIS
LIN {X 0.009,Y -150.370,Z 742.890,A 0.000,B 0.000,C 90.000,E1 160.115} C_DIS
LIN {X 0.027,Y -153.797,Z 742.869,A 0.000,B 0.000,C 90.000,E1 156.485} C_DIS
LIN {X -0.053,Y -157.209,Z 742.849,A 0.000,B 0.000,C 90.000,E1 152.922} C_DIS
LIN {X 0.028,Y -161.373,Z 742.830,A 0.000,B 0.000,C 90.000,E1 149.331} C_DIS
LIN {X 0.039,Y -165.575,Z 742.810,A 0.000,B 0.000,C 90.000,E1 145.801} C_DIS
LIN {X 0.027,Y -170.495,Z 742.791,A 0.000,B 0.000,C 90.000,E1 142.316} C_DIS
LIN {X 0.072,Y -175.375,Z 742.772,A 0.000,B 0.000,C 90.000,E1 138.852} C_DIS
LIN {X -0.066,Y -180.999,Z 742.753,A 0.000,B 0.000,C 90.000,E1 135.486} C_DIS
LIN {X 0.058,Y -186.427,Z 742.734,A 0.000,B 0.000,C 90.000,E1 132.081} C_DIS
LIN {X 0.006,Y -191.505,Z 742.718,A 0.000,B 0.000,C 90.000,E1 129.322} C_DIS
LIN {X -0.079,Y -191.883,Z 742.717,A 0.000,B 0.000,C 90.000,E1 129.116} C_DIS
LIN {X 0.054,Y -290.571,Z 742.717,A 0.000,B 0.000,C 90.000,E1 129.072} C_DIS
LIN {X 0.080,Y -292.644,Z 742.717,A 0.000,B 0.000,C 90.000,E1 129.036} C_DIS
LIN {X 0.135,Y -297.947,Z 742.715,A 0.000,B 0.000,C 90.000,E1 128.749} C_DIS
LIN {X -0.049,Y -301.119,Z 742.714,A 0.000,B 0.000,C 90.000,E1 128.463} C_DIS
LIN {X -0.052,Y -304.734,Z 742.710,A 0.000,B 0.000,C 90.000,E1 127.890} C_DIS
LIN {X 0.144,Y -306.192,Z 742.709,A 0.000,B 0.000,C 90.000,E1 127.523} C_DIS
LIN {X -0.090,Y -307.339,Z 742.707,A 0.000,B 0.000,C 90.000,E1 127.237} C_DIS
LIN {X -0.070,Y -318.148,Z 742.687,A 0.000,B 0.000,C 90.000,E1 123.658} C_DIS
LIN {X -0.119,Y -328.348,Z 742.671,A 0.000,B 0.000,C 90.000,E1 120.797} C_DIS
LIN {X -0.096,Y -339.883,Z 742.655,A 0.000,B 0.000,C 90.000,E1 117.975} C_DIS
LIN {X -0.065,Y -352.861,Z 742.640,A 0.000,B 0.000,C 90.000,E1 115.207} C_DIS
LIN {X 0.147,Y -365.698,Z 742.627,A 0.000,B 0.000,C 90.000,E1 112.770} C_DIS
LIN {X 0.072,Y -379.857,Z 742.614,A 0.000,B 0.000,C 90.000,E1 110.429} C_DIS
LIN {X 0.090,Y -395.440,Z 742.601,A 0.000,B 0.000,C 90.000,E1 108.127} C_DIS
LIN {X -0.014,Y -412.558,Z 742.588,A 0.000,B 0.000,C 90.000,E1 105.898} C_DIS
LIN {X 0.063,Y -431.336,Z 742.576,A 0.000,B 0.000,C 90.000,E1 103.703} C_DIS
LIN {X -0.127,Y -451.349,Z 742.565,A 0.000,B 0.000,C 90.000,E1 101.658} C_DIS
LIN {X 0.055,Y -466.727,Z 742.557,A 0.000,B 0.000,C 90.000,E1 100.197} C_DIS
LIN {X 0.105,Y -469.094,Z 742.555,A 0.000,B 0.000,C 90.000,E1 99.962} C_DIS
LIN {X 0.154,Y -470.889,Z 742.554,A 0.000,B 0.000,C 90.000,E1 99.726} C_DIS
LIN {X -0.072,Y -472.396,Z 742.553,A 0.000,B 0.000,C 90.000,E1 99.500} C_DIS
LIN {X -0.221,Y -473.521,Z 742.551,A 0.000,B 0.000,C 90.000,E1 99.265} C_DIS
LIN {X -0.109,Y -474.865,Z 742.549,A 0.000,B 0.000,C 90.000,E1 98.746} C_DIS
LIN {X 0.082,Y -475.190,Z 742.546,A 0.000,B 0.000,C 90.000,E1 98.219} C_DIS
LIN {X 0.211,Y -474.550,Z 742.543,A 0.000,B 0.000,C 90.000,E1 97.701} C_DIS
LIN {X -0.125,Y -472.847,Z 742.540,A 0.000,B 0.000,C 90.000,E1 97.239} C_DIS
LIN {X 0.201,Y -471.501,Z 742.539,A 0.000,B 0.000,C 90.000,E1 96.947} C_DIS
LIN {X 0.112,Y -452.136,Z 742.522,A 0.000,B 0.000,C 90.000,E1 93.898} C_DIS
LIN {X 0.130,Y -438.786,Z 742.509,A 0.000,B 0.000,C 90.000,E1 91.547} C_DIS
LIN {X 0.073,Y -431.175,Z 742.501,A 0.000,B 0.000,C 90.000,E1 90.229} C_DIS
LIN {X 0.156,Y -420.197,Z 742.491,A 0.000,B 0.000,C 90.000,E1 88.339} C_DIS
LIN {X 0.035,Y -409.170,Z 742.480,A 0.000,B 0.000,C 90.000,E1 86.445} C_DIS
LIN {X 0.134,Y -397.960,Z 742.469,A 0.000,B 0.000,C 90.000,E1 84.489} C_DIS
LIN {X 0.037,Y -385.261,Z 742.457,A 0.000,B 0.000,C 90.000,E1 82.243} C_DIS
LIN {X 0.116,Y -369.910,Z 742.441,A 0.000,B 0.000,C 90.000,E1 79.342} C_DIS
LIN {X -0.050,Y -355.286,Z 742.424,A 0.000,B 0.000,C 90.000,E1 76.408} C_DIS
LIN {X 0.025,Y -345.301,Z 742.413,A 0.000,B 0.000,C 90.000,E1 74.283} C_DIS
LIN {X 0.057,Y -334.153,Z 742.399,A 0.000,B 0.000,C 90.000,E1 71.819} C_DIS
LIN {X 0.082,Y -319.562,Z 742.380,A 0.000,B 0.000,C 90.000,E1 68.358} C_DIS
LIN {X -0.025,Y -308.611,Z 742.364,A 0.000,B 0.000,C 90.000,E1 65.485} C_DIS
LIN {X -0.111,Y -296.765,Z 742.344,A 0.000,B 0.000,C 90.000,E1 61.897} C_DIS
LIN {X 0.002,Y -286.870,Z 742.325,A 0.000,B 0.000,C 90.000,E1 58.535} C_DIS
LIN {X 0.157,Y -277.490,Z 742.306,A 0.000,B 0.000,C 90.000,E1 55.102} C_DIS
LIN {X 0.092,Y -270.200,Z 742.291,A 0.000,B 0.000,C 90.000,E1 52.351} C_DIS
LIN {X -0.013,Y -264.672,Z 742.279,A 0.000,B 0.000,C 90.000,E1 50.275} C_DIS
LIN {X -0.045,Y -259.054,Z 742.268,A 0.000,B 0.000,C 90.000,E1 48.162} C_DIS
LIN {X 0.159,Y -253.361,Z 742.256,A 0.000,B 0.000,C 90.000,E1 45.972} C_DIS
LIN {X -0.108,Y -247.624,Z 742.244,A 0.000,B 0.000,C 90.000,E1 43.866} C_DIS
LIN {X 0.024,Y -239.934,Z 742.227,A 0.000,B 0.000,C 90.000,E1 40.906} C_DIS
LIN {X 0.007,Y -232.294,Z 742.211,A 0.000,B 0.000,C 90.000,E1 37.935} C_DIS
LIN {X 0.134,Y -223.445,Z 742.190,A 0.000,B 0.000,C 90.000,E1 34.119} C_DIS
LIN {X -0.020,Y -216.833,Z 742.173,A 0.000,B 0.000,C 90.000,E1 31.082} C_DIS
LIN {X -0.066,Y -210.920,Z 742.155,A 0.000,B 0.000,C 90.000,E1 27.975} C_DIS
LIN {X 0.000,Y -204.624,Z 742.133,A 0.000,B 0.000,C 90.000,E1 24.003} C_DIS
LIN {X 0.040,Y -200.351,Z 742.116,A 0.000,B 0.000,C 90.000,E1 20.791} C_DIS
LIN {X 0.094,Y -196.088,Z 742.093,A 0.000,B 0.000,C 90.000,E1 16.732} C_DIS
LIN {X -0.072,Y -192.361,Z 742.066,A 0.000,B 0.000,C 90.000,E1 11.883} C_DIS
LIN {X -0.004,Y -189.724,Z 742.029,A 0.000,B 0.000,C 90.000,E1 5.277} C_DIS
LIN {X 0.076,Y -190.903,Z 741.970,A 0.000,B 0.000,C 90.000,E1 354.552} C_DIS
LIN {X 0.012,Y -193.735,Z 741.942,A 0.000,B 0.000,C 90.000,E1 349.634} C_DIS
LIN {X 0.104,Y -197.272,Z 741.920,A 0.000,B 0.000,C 90.000,E1 345.519} C_DIS
LIN {X -0.056,Y -201.679,Z 741.897,A 0.000,B 0.000,C 90.000,E1 341.511} C_DIS
LIN {X -0.015,Y -207.180,Z 741.875,A 0.000,B 0.000,C 90.000,E1 337.486} C_DIS
LIN {X 0.022,Y -213.548,Z 741.853,A 0.000,B 0.000,C 90.000,E1 333.512} C_DIS
LIN {X 0.011,Y -219.153,Z 741.835,A 0.000,B 0.000,C 90.000,E1 330.383} C_DIS
LIN {X 0.092,Y -226.698,Z 741.814,A 0.000,B 0.000,C 90.000,E1 326.501} C_DIS
LIN {X -0.075,Y -233.230,Z 741.797,A 0.000,B 0.000,C 90.000,E1 323.497} C_DIS
LIN {X -0.074,Y -241.875,Z 741.776,A 0.000,B 0.000,C 90.000,E1 319.747} C_DIS
LIN {X -0.030,Y -251.488,Z 741.756,A 0.000,B 0.000,C 90.000,E1 316.053} C_DIS
LIN {X 0.126,Y -260.970,Z 741.738,A 0.000,B 0.000,C 90.000,E1 312.771} C_DIS
LIN {X -0.072,Y -272.443,Z 741.718,A 0.000,B 0.000,C 90.000,E1 309.277} C_DIS
LIN {X 0.048,Y -283.854,Z 741.701,A 0.000,B 0.000,C 90.000,E1 306.137} C_DIS
LIN {X -0.062,Y -292.057,Z 741.689,A 0.000,B 0.000,C 90.000,E1 304.119} C_DIS
LIN {X -0.131,Y -305.660,Z 741.673,A 0.000,B 0.000,C 90.000,E1 301.131} C_DIS
LIN {X 0.080,Y -319.076,Z 741.658,A 0.000,B 0.000,C 90.000,E1 298.487} C_DIS
LIN {X -0.137,Y -335.440,Z 741.642,A 0.000,B 0.000,C 90.000,E1 295.668} C_DIS
LIN {X -0.176,Y -353.122,Z 741.627,A 0.000,B 0.000,C 90.000,E1 292.898} C_DIS
LIN {X -0.080,Y -369.902,Z 741.614,A 0.000,B 0.000,C 90.000,E1 290.482} C_DIS
LIN {X -0.168,Y -390.578,Z 741.599,A 0.000,B 0.000,C 90.000,E1 287.873} C_DIS
LIN {X 0.189,Y -407.344,Z 741.588,A 0.000,B 0.000,C 90.000,E1 285.843} C_DIS
LIN {X 0.035,Y -419.193,Z 741.581,A 0.000,B 0.000,C 90.000,E1 284.481} C_DIS
LIN {X 0.059,Y -430.803,Z 741.573,A 0.000,B 0.000,C 90.000,E1 283.119} C_DIS
LIN {X 0.153,Y -441.969,Z 741.565,A 0.000,B 0.000,C 90.000,E1 281.771} C_DIS
LIN {X 0.091,Y -450.416,Z 741.560,A 0.000,B 0.000,C 90.000,E1 280.725} C_DIS
LIN {X -0.225,Y -462.554,Z 741.551,A 0.000,B 0.000,C 90.000,E1 279.208} C_DIS
LIN {X -0.046,Y -470.467,Z 741.545,A 0.000,B 0.000,C 90.000,E1 278.163} C_DIS
LIN {X -0.100,Y -475.971,Z 741.541,A 0.000,B 0.000,C 90.000,E1 277.409} C_DIS
LIN {X -0.171,Y -480.804,Z 741.537,A 0.000,B 0.000,C 90.000,E1 276.663} C_DIS
LIN {X -0.139,Y -484.901,Z 741.533,A 0.000,B 0.000,C 90.000,E1 275.910} C_DIS
LIN {X 0.044,Y -487.223,Z 741.530,A 0.000,B 0.000,C 90.000,E1 275.391} C_DIS
LIN {X 0.079,Y -489.956,Z 741.526,A 0.000,B 0.000,C 90.000,E1 274.645} C_DIS
LIN {X -0.237,Y -491.276,Z 741.523,A 0.000,B 0.000,C 90.000,E1 274.188} C_DIS
LIN {X -0.017,Y -492.207,Z 741.520,A 0.000,B 0.000,C 90.000,E1 273.669} C_DIS
LIN {X 0.181,Y -492.707,Z 741.518,A 0.000,B 0.000,C 90.000,E1 273.154} C_DIS
LIN {X -0.082,Y -492.827,Z 741.515,A 0.000,B 0.000,C 90.000,E1 272.694} C_DIS
LIN {X 0.128,Y -492.481,Z 741.512,A 0.000,B 0.000,C 90.000,E1 272.178} C_DIS
LIN {X -0.137,Y -491.760,Z 741.509,A 0.000,B 0.000,C 90.000,E1 271.718} C_DIS
LIN {X 0.070,Y -490.564,Z 741.507,A 0.000,B 0.000,C 90.000,E1 271.203} C_DIS
LIN {X -0.215,Y -488.942,Z 741.504,A 0.000,B 0.000,C 90.000,E1 270.745} C_DIS
LIN {X -0.016,Y -486.763,Z 741.501,A 0.000,B 0.000,C 90.000,E1 270.229} C_DIS
LIN {X 0.166,Y -483.966,Z 741.499,A 0.000,B 0.000,C 90.000,E1 269.714} C_DIS
LIN {X -0.149,Y -480.424,Z 741.496,A 0.000,B 0.000,C 90.000,E1 269.255} C_DIS
LIN {X -0.002,Y -475.992,Z 741.493,A 0.000,B 0.000,C 90.000,E1 268.740} C_DIS
LIN {X 0.119,Y -470.395,Z 741.490,A 0.000,B 0.000,C 90.000,E1 268.224} C_DIS
LIN {X 0.182,Y -467.521,Z 741.489,A 0.000,B 0.000,C 90.000,E1 267.993} C_DIS
LIN {X 0.076,Y -461.169,Z 741.487,A 0.000,B 0.000,C 90.000,E1 267.593} C_DIS
LIN {X 0.013,Y -454.345,Z 741.485,A 0.000,B 0.000,C 90.000,E1 267.249} C_DIS
LIN {X 0.099,Y -450.561,Z 741.484,A 0.000,B 0.000,C 90.000,E1 267.078} C_DIS
LIN {X -0.102,Y -442.992,Z 741.482,A 0.000,B 0.000,C 90.000,E1 266.846} C_DIS
LIN {X 0.096,Y -434.355,Z 741.481,A 0.000,B 0.000,C 90.000,E1 266.617} C_DIS
LIN {X 0.020,Y -430.088,Z 741.481,A 0.000,B 0.000,C 90.000,E1 266.560} C_DIS
LIN {X -0.198,Y -419.951,Z 741.480,A 0.000,B 0.000,C 90.000,E1 266.502} C_DIS
LIN {X 0.065,Y -180.946,Z 741.480,A 0.000,B 0.000,C 90.000,E1 266.445} C_DIS
LIN {X 0.025,Y -180.780,Z 741.471,A 0.000,B 0.000,C 90.000,E1 264.723} C_DIS
LIN {X -0.080,Y -178.876,Z 741.443,A 0.000,B 0.000,C 90.000,E1 259.690} C_DIS
LIN {X -0.004,Y -175.919,Z 741.414,A 0.000,B 0.000,C 90.000,E1 254.574} C_DIS
LIN {X 0.053,Y -174.614,Z 741.405,A 0.000,B 0.000,C 90.000,E1 252.851} C_DIS
LIN {X -0.022,Y -171.595,Z 741.381,A 0.000,B 0.000,C 90.000,E1 248.592} C_DIS
LIN {X -0.032,Y -167.818,Z 741.357,A 0.000,B 0.000,C 90.000,E1 244.280} C_DIS
LIN {X -0.016,Y -166.540,Z 741.347,A 0.000,B 0.000,C 90.000,E1 242.538} C_DIS
LIN {X -0.104,Y -162.537,Z 741.323,A 0.000,B 0.000,C 90.000,E1 238.201} C_DIS
LIN {X -0.044,Y -161.214,Z 741.313,A 0.000,B 0.000,C 90.000,E1 236.421} C_DIS
LIN {X -0.008,Y -157.221,Z 741.289,A 0.000,B 0.000,C 90.000,E1 231.984} C_DIS
LIN {X 0.015,Y -155.948,Z 741.279,A 0.000,B 0.000,C 90.000,E1 230.194} C_DIS
LIN {X -0.026,Y -152.200,Z 741.254,A 0.000,B 0.000,C 90.000,E1 225.729} C_DIS
LIN {X -0.004,Y -150.445,Z 741.239,A 0.000,B 0.000,C 90.000,E1 223.014} C_DIS
LIN {X 0.022,Y -147.171,Z 741.214,A 0.000,B 0.000,C 90.000,E1 218.463} C_DIS
LIN {X -0.011,Y -145.188,Z 741.193,A 0.000,B 0.000,C 90.000,E1 214.818} C_DIS
LIN {X 0.024,Y -142.331,Z 741.163,A 0.000,B 0.000,C 90.000,E1 209.283} C_DIS
LIN {X -0.047,Y -141.720,Z 741.152,A 0.000,B 0.000,C 90.000,E1 207.462} C_DIS
LIN {X 0.065,Y -139.476,Z 741.116,A 0.000,B 0.000,C 90.000,E1 200.918} C_DIS
LIN {X -0.075,Y -138.974,Z 741.101,A 0.000,B 0.000,C 90.000,E1 198.181} C_DIS
LIN {X 0.046,Y -138.331,Z 741.054,A 0.000,B 0.000,C 90.000,E1 189.726} C_DIS
LIN {X 0.049,Y -139.434,Z 741.007,A 0.000,B 0.000,C 90.000,E1 181.318} C_DIS
LIN {X -0.011,Y -140.962,Z 740.976,A 0.000,B 0.000,C 90.000,E1 175.755} C_DIS
LIN {X -0.061,Y -142.717,Z 740.956,A 0.000,B 0.000,C 90.000,E1 172.064} C_DIS
LIN {X 0.038,Y -145.097,Z 740.930,A 0.000,B 0.000,C 90.000,E1 167.409} C_DIS
LIN {X 0.033,Y -147.722,Z 740.910,A 0.000,B 0.000,C 90.000,E1 163.740} C_DIS
LIN {X -0.026,Y -150.380,Z 740.889,A 0.000,B 0.000,C 90.000,E1 160.115} C_DIS
LIN {X -0.008,Y -153.811,Z 740.869,A 0.000,B 0.000,C 90.000,E1 156.485} C_DIS
LIN {X 0.052,Y -157.222,Z 740.849,A 0.000,B 0.000,C 90.000,E1 152.871} C_DIS
LIN {X -0.007,Y -161.389,Z 740.830,A 0.000,B 0.000,C 90.000,E1 149.331} C_DIS
LIN {X 0.003,Y -165.591,Z 740.810,A 0.000,B 0.000,C 90.000,E1 145.801} C_DIS
LIN {X -0.011,Y -170.513,Z 740.791,A 0.000,B 0.000,C 90.000,E1 142.316} C_DIS
LIN {X 0.034,Y -175.393,Z 740.771,A 0.000,B 0.000,C 90.000,E1 138.852} C_DIS
LIN {X -0.104,Y -181.017,Z 740.753,A 0.000,B 0.000,C 90.000,E1 135.486} C_DIS
LIN {X 0.019,Y -186.448,Z 740.734,A 0.000,B 0.000,C 90.000,E1 132.081} C_DIS
LIN {X -0.032,Y -191.523,Z 740.718,A 0.000,B 0.000,C 90.000,E1 129.322} C_DIS
LIN {X -0.036,Y -191.863,Z 740.717,A 0.000,B 0.000,C 90.000,E1 129.116} C_DIS
LIN {X -0.085,Y -290.954,Z 740.717,A 0.000,B 0.000,C 90.000,E1 129.116} C_DIS
LIN {X 0.051,Y -292.135,Z 740.717,A 0.000,B 0.000,C 90.000,E1 129.072} C_DIS
LIN {X 0.063,Y -296.077,Z 740.716,A 0.000,B 0.000,C 90.000,E1 128.910} C_DIS
LIN {X 0.073,Y -298.263,Z 740.715,A 0.000,B 0.000,C 90.000,E1 128.749} C_DIS
LIN {X -0.053,Y -302.146,Z 740.713,A 0.000,B 0.000,C 90.000,E1 128.338} C_DIS
LIN {X 0.012,Y -304.051,Z 740.711,A 0.000,B 0.000,C 90.000,E1 128.016} C_DIS
LIN {X -0.111,Y -305.550,Z 740.709,A 0.000,B 0.000,C 90.000,E1 127.729} C_DIS
LIN {X 0.093,Y -306.812,Z 740.708,A 0.000,B 0.000,C 90.000,E1 127.363} C_DIS
LIN {X -0.104,Y -318.675,Z 740.686,A 0.000,B 0.000,C 90.000,E1 123.499} C_DIS
LIN {X 0.132,Y -328.948,Z 740.670,A 0.000,B 0.000,C 90.000,E1 120.590} C_DIS
LIN {X 0.177,Y -340.563,Z 740.654,A 0.000,B 0.000,C 90.000,E1 117.769} C_DIS
LIN {X 0.081,Y -353.627,Z 740.639,A 0.000,B 0.000,C 90.000,E1 115.027} C_DIS
LIN {X -0.015,Y -366.545,Z 740.626,A 0.000,B 0.000,C 90.000,E1 112.642} C_DIS
LIN {X -0.077,Y -380.793,Z 740.613,A 0.000,B 0.000,C 90.000,E1 110.301} C_DIS
LIN {X -0.047,Y -396.470,Z 740.600,A 0.000,B 0.000,C 90.000,E1 108.000} C_DIS
LIN {X 0.149,Y -413.691,Z 740.588,A 0.000,B 0.000,C 90.000,E1 105.733} C_DIS
LIN {X -0.146,Y -432.581,Z 740.575,A 0.000,B 0.000,C 90.000,E1 103.592} C_DIS
LIN {X -0.157,Y -452.632,Z 740.564,A 0.000,B 0.000,C 90.000,E1 101.535} C_DIS
LIN {X 0.081,Y -468.012,Z 740.556,A 0.000,B 0.000,C 90.000,E1 100.074} C_DIS
LIN {X 0.021,Y -470.098,Z 740.555,A 0.000,B 0.000,C 90.000,E1 99.849} C_DIS
LIN {X 0.042,Y -471.683,Z 740.553,A 0.000,B 0.000,C 90.000,E1 99.613} C_DIS
LIN {X -0.104,Y -472.992,Z 740.552,A 0.000,B 0.000,C 90.000,E1 99.378} C_DIS
LIN {X 0.141,Y -473.958,Z 740.551,A 0.000,B 0.000,C 90.000,E1 99.095} C_DIS
LIN {X -0.138,Y -475.041,Z 740.548,A 0.000,B 0.000,C 90.000,E1 98.624} C_DIS
LIN {X -0.014,Y -475.132,Z 740.545,A 0.000,B 0.000,C 90.000,E1 98.106} C_DIS
LIN {X 0.117,Y -474.249,Z 740.542,A 0.000,B 0.000,C 90.000,E1 97.587} C_DIS
LIN {X -0.219,Y -472.250,Z 740.539,A 0.000,B 0.000,C 90.000,E1 97.125} C_DIS
LIN {X 0.017,Y -465.704,Z 740.534,A 0.000,B 0.000,C 90.000,E1 96.087} C_DIS
LIN {X 0.214,Y -449.882,Z 740.520,A 0.000,B 0.000,C 90.000,E1 93.498} C_DIS
LIN {X 0.005,Y -438.092,Z 740.508,A 0.000,B 0.000,C 90.000,E1 91.432} C_DIS
LIN {X -0.059,Y -430.460,Z 740.501,A 0.000,B 0.000,C 90.000,E1 90.115} C_DIS
LIN {X 0.011,Y -419.503,Z 740.490,A 0.000,B 0.000,C 90.000,E1 88.224} C_DIS
LIN {X -0.121,Y -408.450,Z 740.479,A 0.000,B 0.000,C 90.000,E1 86.331} C_DIS
LIN {X -0.033,Y -397.253,Z 740.469,A 0.000,B 0.000,C 90.000,E1 84.375} C_DIS
LIN {X -0.145,Y -384.587,Z 740.456,A 0.000,B 0.000,C 90.000,E1 82.129} C_DIS
LIN {X -0.017,Y -370.777,Z 740.442,A 0.000,B 0.000,C 90.000,E1 79.511} C_DIS
LIN {X -0.180,Y -357.537,Z 740.427,A 0.000,B 0.000,C 90.000,E1 76.881} C_DIS
LIN {X -0.053,Y -347.577,Z 740.415,A 0.000,B 0.000,C 90.000,E1 74.755} C_DIS
LIN {X -0.069,Y -334.987,Z 740.400,A 0.000,B 0.000,C 90.000,E1 72.000} C_DIS
LIN {X -0.014,Y -320.359,Z 740.381,A 0.000,B 0.000,C 90.000,E1 68.539} C_DIS
LIN {X -0.088,Y -309.385,Z 740.365,A 0.000,B 0.000,C 90.000,E1 65.665} C_DIS
LIN {X 0.102,Y -298.551,Z 740.347,A 0.000,B 0.000,C 90.000,E1 62.359} C_DIS
LIN {X -0.134,Y -288.595,Z 740.328,A 0.000,B 0.000,C 90.000,E1 59.076} C_DIS
LIN {X -0.076,Y -279.183,Z 740.309,A 0.000,B 0.000,C 90.000,E1 55.674} C_DIS
LIN {X -0.096,Y -271.929,Z 740.294,A 0.000,B 0.000,C 90.000,E1 52.924} C_DIS
LIN {X 0.043,Y -266.452,Z 740.282,A 0.000,B 0.000,C 90.000,E1 50.803} C_DIS
LIN {X 0.042,Y -260.868,Z 740.271,A 0.000,B 0.000,C 90.000,E1 48.690} C_DIS
LIN {X 0.157,Y -253.293,Z 740.255,A 0.000,B 0.000,C 90.000,E1 45.810} C_DIS
LIN {X -0.112,Y -247.558,Z 740.243,A 0.000,B 0.000,C 90.000,E1 43.704} C_DIS
LIN {X 0.018,Y -239.849,Z 740.226,A 0.000,B 0.000,C 90.000,E1 40.744} C_DIS
LIN {X -0.149,Y -232.202,Z 740.210,A 0.000,B 0.000,C 90.000,E1 37.810} C_DIS
LIN {X -0.012,Y -223.338,Z 740.189,A 0.000,B 0.000,C 90.000,E1 33.992} C_DIS
LIN {X -0.050,Y -216.739,Z 740.172,A 0.000,B 0.000,C 90.000,E1 30.924} C_DIS
LIN {X 0.081,Y -210.842,Z 740.154,A 0.000,B 0.000,C 90.000,E1 27.769} C_DIS
LIN {X 0.050,Y -204.550,Z 740.132,A 0.000,B 0.000,C 90.000,E1 23.823} C_DIS
LIN {X 0.089,Y -200.305,Z 740.115,A 0.000,B 0.000,C 90.000,E1 20.610} C_DIS
LIN {X -0.102,Y -196.080,Z 740.092,A 0.000,B 0.000,C 90.000,E1 16.622} C_DIS
LIN {X -0.068,Y -192.392,Z 740.065,A 0.000,B 0.000,C 90.000,E1 11.715} C_DIS
LIN {X 0.011,Y -189.783,Z 740.028,A 0.000,B 0.000,C 90.000,E1 5.106} C_DIS
LIN {X 0.079,Y -190.977,Z 739.970,A 0.000,B 0.000,C 90.000,E1 354.552} C_DIS
LIN {X 0.018,Y -193.820,Z 739.942,A 0.000,B 0.000,C 90.000,E1 349.634} C_DIS
LIN {X 0.113,Y -197.367,Z 739.920,A 0.000,B 0.000,C 90.000,E1 345.519} C_DIS
LIN {X -0.043,Y -201.797,Z 739.897,A 0.000,B 0.000,C 90.000,E1 341.511} C_DIS
LIN {X 0.001,Y -207.289,Z 739.875,A 0.000,B 0.000,C 90.000,E1 337.486} C_DIS
LIN {X 0.042,Y -213.672,Z 739.853,A 0.000,B 0.000,C 90.000,E1 333.512} C_DIS
LIN {X -0.002,Y -220.698,Z 739.831,A 0.000,B 0.000,C 90.000,E1 329.616} C_DIS
LIN {X 0.047,Y -228.362,Z 739.810,A 0.000,B 0.000,C 90.000,E1 325.754} C_DIS
LIN {X 0.053,Y -234.954,Z 739.793,A 0.000,B 0.000,C 90.000,E1 322.718} C_DIS
LIN {X -0.042,Y -241.907,Z 739.776,A 0.000,B 0.000,C 90.000,E1 319.747} C_DIS
LIN {X 0.005,Y -251.512,Z 739.756,A 0.000,B 0.000,C 90.000,E1 316.053} C_DIS
LIN {X -0.029,Y -260.990,Z 739.738,A 0.000,B 0.000,C 90.000,E1 312.813} C_DIS
LIN {X -0.033,Y -272.457,Z 739.718,A 0.000,B 0.000,C 90.000,E1 309.277} C_DIS
LIN {X 0.045,Y -285.183,Z 739.699,A 0.000,B 0.000,C 90.000,E1 305.804} C_DIS
LIN {X -0.049,Y -294.987,Z 739.686,A 0.000,B 0.000,C 90.000,E1 303.452} C_DIS
LIN {X -0.025,Y -308.901,Z 739.669,A 0.000,B 0.000,C 90.000,E1 300.463} C_DIS
LIN {X 0.043,Y -320.867,Z 739.657,A 0.000,B 0.000,C 90.000,E1 298.180} C_DIS
LIN {X 0.011,Y -339.221,Z 739.639,A 0.000,B 0.000,C 90.000,E1 295.027} C_DIS
LIN {X -0.097,Y -355.110,Z 739.625,A 0.000,B 0.000,C 90.000,E1 292.589} C_DIS
LIN {X 0.052,Y -372.002,Z 739.612,A 0.000,B 0.000,C 90.000,E1 290.174} C_DIS
LIN {X -0.084,Y -392.789,Z 739.598,A 0.000,B 0.000,C 90.000,E1 287.583} C_DIS
LIN {X -0.152,Y -407.159,Z 739.588,A 0.000,B 0.000,C 90.000,E1 285.898} C_DIS
LIN {X 0.085,Y -418.987,Z 739.581,A 0.000,B 0.000,C 90.000,E1 284.481} C_DIS
LIN {X 0.108,Y -430.597,Z 739.573,A 0.000,B 0.000,C 90.000,E1 283.119} C_DIS
LIN {X 0.200,Y -441.749,Z 739.566,A 0.000,B 0.000,C 90.000,E1 281.771} C_DIS
LIN {X -0.061,Y -452.243,Z 739.558,A 0.000,B 0.000,C 90.000,E1 280.489} C_DIS
LIN {X 0.103,Y -464.327,Z 739.550,A 0.000,B 0.000,C 90.000,E1 278.916} C_DIS
LIN {X -0.226,Y -472.155,Z 739.544,A 0.000,B 0.000,C 90.000,E1 277.936} C_DIS
LIN {X 0.204,Y -477.446,Z 739.540,A 0.000,B 0.000,C 90.000,E1 277.125} C_DIS
LIN {X 0.212,Y -482.062,Z 739.536,A 0.000,B 0.000,C 90.000,E1 276.372} C_DIS
LIN {X 0.203,Y -485.910,Z 739.531,A 0.000,B 0.000,C 90.000,E1 275.625} C_DIS
LIN {X -0.090,Y -488.036,Z 739.529,A 0.000,B 0.000,C 90.000,E1 275.163} C_DIS
LIN {X 0.114,Y -489.763,Z 739.526,A 0.000,B 0.000,C 90.000,E1 274.645} C_DIS
LIN {X -0.203,Y -491.083,Z 739.523,A 0.000,B 0.000,C 90.000,E1 274.188} C_DIS
LIN {X 0.016,Y -491.986,Z 739.520,A 0.000,B 0.000,C 90.000,E1 273.669} C_DIS
LIN {X 0.212,Y -492.514,Z 739.518,A 0.000,B 0.000,C 90.000,E1 273.154} C_DIS
LIN {X -0.051,Y -492.605,Z 739.515,A 0.000,B 0.000,C 90.000,E1 272.694} C_DIS
LIN {X 0.157,Y -492.290,Z 739.512,A 0.000,B 0.000,C 90.000,E1 272.178} C_DIS
LIN {X -0.109,Y -491.566,Z 739.509,A 0.000,B 0.000,C 90.000,E1 271.718} C_DIS
LIN {X 0.097,Y -490.418,Z 739.507,A 0.000,B 0.000,C 90.000,E1 271.203} C_DIS
LIN {X -0.189,Y -488.812,Z 739.504,A 0.000,B 0.000,C 90.000,E1 270.745} C_DIS
LIN {X 0.008,Y -486.678,Z 739.501,A 0.000,B 0.000,C 90.000,E1 270.229} C_DIS
LIN {X 0.195,Y -483.896,Z 739.499,A 0.000,B 0.000,C 90.000,E1 269.714} C_DIS
LIN {X -0.121,Y -480.443,Z 739.496,A 0.000,B 0.000,C 90.000,E1 269.255} C_DIS
LIN {X 0.027,Y -476.016,Z 739.493,A 0.000,B 0.000,C 90.000,E1 268.740} C_DIS
LIN {X 0.147,Y -470.512,Z 739.490,A 0.000,B 0.000,C 90.000,E1 268.224} C_DIS
LIN {X 0.213,Y -464.278,Z 739.488,A 0.000,B 0.000,C 90.000,E1 267.764} C_DIS
LIN {X 0.050,Y -461.250,Z 739.487,A 0.000,B 0.000,C 90.000,E1 267.593} C_DIS
LIN {X -0.021,Y -454.463,Z 739.485,A 0.000,B 0.000,C 90.000,E1 267.249} C_DIS
LIN {X -0.044,Y -447.193,Z 739.483,A 0.000,B 0.000,C 90.000,E1 266.963} C_DIS
LIN {X -0.008,Y -439.481,Z 739.482,A 0.000,B 0.000,C 90.000,E1 266.731} C_DIS
LIN {X 0.026,Y -430.880,Z 739.481,A 0.000,B 0.000,C 90.000,E1 266.560} C_DIS
LIN {X 0.209,Y -421.814,Z 739.480,A 0.000,B 0.000,C 90.000,E1 266.445} C_DIS
LIN {X 0.131,Y -419.441,Z 739.480,A 0.000,B 0.000,C 90.000,E1 266.445} C_DIS
LIN {X 0.022,Y -180.945,Z 739.480,A 0.000,B 0.000,C 90.000,E1 266.445} C_DIS
LIN {X 0.005,Y -180.777,Z 739.471,A 0.000,B 0.000,C 90.000,E1 264.723} C_DIS
LIN {X 0.076,Y -178.873,Z 739.443,A 0.000,B 0.000,C 90.000,E1 259.634} C_DIS
LIN {X -0.024,Y -175.916,Z 739.414,A 0.000,B 0.000,C 90.000,E1 254.574} C_DIS
LIN {X 0.032,Y -174.608,Z 739.405,A 0.000,B 0.000,C 90.000,E1 252.851} C_DIS
LIN {X -0.041,Y -171.590,Z 739.381,A 0.000,B 0.000,C 90.000,E1 248.592} C_DIS
LIN {X -0.052,Y -167.813,Z 739.357,A 0.000,B 0.000,C 90.000,E1 244.280} C_DIS
LIN {X -0.035,Y -166.534,Z 739.347,A 0.000,B 0.000,C 90.000,E1 242.538} C_DIS
LIN {X 0.015,Y -162.532,Z 739.323,A 0.000,B 0.000,C 90.000,E1 238.152} C_DIS
LIN {X -0.063,Y -161.207,Z 739.313,A 0.000,B 0.000,C 90.000,E1 236.421} C_DIS
LIN {X -0.027,Y -157.216,Z 739.289,A 0.000,B 0.000,C 90.000,E1 231.984} C_DIS
LIN {X -0.004,Y -155.943,Z 739.279,A 0.000,B 0.000,C 90.000,E1 230.194} C_DIS
LIN {X -0.044,Y -152.195,Z 739.254,A 0.000,B 0.000,C 90.000,E1 225.729} C_DIS
LIN {X -0.024,Y -150.441,Z 739.239,A 0.000,B 0.000,C 90.000,E1 223.014} C_DIS
LIN {X 0.004,Y -147.168,Z 739.214,A 0.000,B 0.000,C 90.000,E1 218.463} C_DIS
LIN {X -0.028,Y -145.183,Z 739.193,A 0.000,B 0.000,C 90.000,E1 214.818} C_DIS
LIN {X 0.006,Y -142.328,Z 739.163,A 0.000,B 0.000,C 90.000,E1 209.283} C_DIS
LIN {X 0.001,Y -141.718,Z 739.152,A 0.000,B 0.000,C 90.000,E1 207.436} C_DIS
LIN {X 0.049,Y -139.475,Z 739.116,A 0.000,B 0.000,C 90.000,E1 200.918} C_DIS
LIN {X 0.040,Y -138.972,Z 739.101,A 0.000,B 0.000,C 90.000,E1 198.127} C_DIS
LIN {X 0.028,Y -138.330,Z 739.054,A 0.000,B 0.000,C 90.000,E1 189.726} C_DIS
LIN {X 0.032,Y -139.436,Z 739.007,A 0.000,B 0.000,C 90.000,E1 181.318} C_DIS
LIN {X -0.029,Y -140.965,Z 738.976,A 0.000,B 0.000,C 90.000,E1 175.755} C_DIS
LIN {X 0.063,Y -142.721,Z 738.956,A 0.000,B 0.000,C 90.000,E1 172.008} C_DIS
LIN {X 0.021,Y -145.101,Z 738.930,A 0.000,B 0.000,C 90.000,E1 167.409} C_DIS
LIN {X 0.016,Y -147.726,Z 738.910,A 0.000,B 0.000,C 90.000,E1 163.740} C_DIS
LIN {X -0.044,Y -150.386,Z 738.889,A 0.000,B 0.000,C 90.000,E1 160.115} C_DIS
LIN {X -0.027,Y -153.818,Z 738.869,A 0.000,B 0.000,C 90.000,E1 156.485} C_DIS
LIN {X 0.033,Y -157.230,Z 738.849,A 0.000,B 0.000,C 90.000,E1 152.871} C_DIS
LIN {X -0.027,Y -161.397,Z 738.830,A 0.000,B 0.000,C 90.000,E1 149.331} C_DIS
LIN {X -0.016,Y -165.599,Z 738.810,A 0.000,B 0.000,C 90.000,E1 145.801} C_DIS
LIN {X -0.030,Y -170.524,Z 738.791,A 0.000,B 0.000,C 90.000,E1 142.316} C_DIS
LIN {X 0.013,Y -175.403,Z 738.771,A 0.000,B 0.000,C 90.000,E1 138.852} C_DIS
LIN {X 0.004,Y -181.028,Z 738.753,A 0.000,B 0.000,C 90.000,E1 135.445} C_DIS
LIN {X -0.002,Y -186.459,Z 738.734,A 0.000,B 0.000,C 90.000,E1 132.081} C_DIS
LIN {X 0.095,Y -191.533,Z 738.718,A 0.000,B 0.000,C 90.000,E1 129.277} C_DIS
LIN {X 0.024,Y -191.833,Z 738.717,A 0.000,B 0.000,C 90.000,E1 129.116} C_DIS
LIN {X 0.007,Y -290.892,Z 738.717,A 0.000,B 0.000,C 90.000,E1 129.116} C_DIS
LIN {X 0.022,Y -293.007,Z 738.717,A 0.000,B 0.000,C 90.000,E1 129.072} C_DIS
LIN {X 0.040,Y -298.477,Z 738.715,A 0.000,B 0.000,C 90.000,E1 128.749} C_DIS
LIN {X 0.092,Y -301.690,Z 738.713,A 0.000,B 0.000,C 90.000,E1 128.382} C_DIS
LIN {X -0.019,Y -303.671,Z 738.712,A 0.000,B 0.000,C 90.000,E1 128.096} C_DIS
LIN {X -0.130,Y -305.224,Z 738.710,A 0.000,B 0.000,C 90.000,E1 127.810} C_DIS
LIN {X 0.073,Y -306.540,Z 738.708,A 0.000,B 0.000,C 90.000,E1 127.443} C_DIS
LIN {X 0.152,Y -314.260,Z 738.694,A 0.000,B 0.000,C 90.000,E1 124.818} C_DIS
LIN {X -0.190,Y -325.087,Z 738.676,A 0.000,B 0.000,C 90.000,E1 121.671} C_DIS
LIN {X -0.102,Y -336.211,Z 738.660,A 0.000,B 0.000,C 90.000,E1 118.821} C_DIS
LIN {X -0.016,Y -348.738,Z 738.645,A 0.000,B 0.000,C 90.000,E1 116.027} C_DIS
LIN {X 0.087,Y -361.147,Z 738.631,A 0.000,B 0.000,C 90.000,E1 113.590} C_DIS
LIN {X 0.040,Y -374.845,Z 738.618,A 0.000,B 0.000,C 90.000,E1 111.227} C_DIS
LIN {X 0.058,Y -389.931,Z 738.605,A 0.000,B 0.000,C 90.000,E1 108.906} C_DIS
LIN {X -0.183,Y -406.513,Z 738.593,A 0.000,B 0.000,C 90.000,E1 106.677} C_DIS
LIN {X 0.154,Y -424.713,Z 738.580,A 0.000,B 0.000,C 90.000,E1 104.426} C_DIS
LIN {X 0.205,Y -444.423,Z 738.568,A 0.000,B 0.000,C 90.000,E1 102.299} C_DIS
LIN {X 0.040,Y -464.811,Z 738.558,A 0.000,B 0.000,C 90.000,E1 100.366} C_DIS
LIN {X -0.028,Y -467.411,Z 738.556,A 0.000,B 0.000,C 90.000,E1 100.141} C_DIS
LIN {X 0.027,Y -469.620,Z 738.555,A 0.000,B 0.000,C 90.000,E1 99.905} C_DIS
LIN {X 0.082,Y -471.291,Z 738.554,A 0.000,B 0.000,C 90.000,E1 99.670} C_DIS
LIN {X -0.143,Y -472.701,Z 738.552,A 0.000,B 0.000,C 90.000,E1 99.443} C_DIS
LIN {X 0.178,Y -473.748,Z 738.551,A 0.000,B 0.000,C 90.000,E1 99.151} C_DIS
LIN {X -0.103,Y -474.966,Z 738.548,A 0.000,B 0.000,C 90.000,E1 98.681} C_DIS
LIN {X 0.018,Y -475.179,Z 738.545,A 0.000,B 0.000,C 90.000,E1 98.163} C_DIS
LIN {X 0.147,Y -474.425,Z 738.543,A 0.000,B 0.000,C 90.000,E1 97.644} C_DIS
LIN {X -0.189,Y -472.583,Z 738.540,A 0.000,B 0.000,C 90.000,E1 97.182} C_DIS
LIN {X -0.060,Y -469.473,Z 738.537,A 0.000,B 0.000,C 90.000,E1 96.663} C_DIS
LIN {X 0.041,Y -451.781,Z 738.521,A 0.000,B 0.000,C 90.000,E1 93.841} C_DIS
LIN {X 0.054,Y -438.478,Z 738.508,A 0.000,B 0.000,C 90.000,E1 91.489} C_DIS
LIN {X -0.005,Y -430.880,Z 738.501,A 0.000,B 0.000,C 90.000,E1 90.172} C_DIS
LIN {X 0.195,Y -418.390,Z 738.489,A 0.000,B 0.000,C 90.000,E1 87.993} C_DIS
LIN {X -0.051,Y -408.894,Z 738.480,A 0.000,B 0.000,C 90.000,E1 86.388} C_DIS
LIN {X 0.045,Y -397.727,Z 738.469,A 0.000,B 0.000,C 90.000,E1 84.432} C_DIS
LIN {X -0.020,Y -383.502,Z 738.455,A 0.000,B 0.000,C 90.000,E1 81.894} C_DIS
LIN {X 0.017,Y -369.760,Z 738.440,A 0.000,B 0.000,C 90.000,E1 79.285} C_DIS
LIN {X -0.109,Y -356.577,Z 738.426,A 0.000,B 0.000,C 90.000,E1 76.645} C_DIS
LIN {X 0.000,Y -346.636,Z 738.414,A 0.000,B 0.000,C 90.000,E1 74.519} C_DIS
LIN {X -0.051,Y -334.092,Z 738.399,A 0.000,B 0.000,C 90.000,E1 71.764} C_DIS
LIN {X 0.089,Y -319.565,Z 738.379,A 0.000,B 0.000,C 90.000,E1 68.284} C_DIS
LIN {X -0.009,Y -308.732,Z 738.363,A 0.000,B 0.000,C 90.000,E1 65.409} C_DIS
LIN {X -0.081,Y -297.003,Z 738.343,A 0.000,B 0.000,C 90.000,E1 61.820} C_DIS
LIN {X 0.044,Y -287.200,Z 738.325,A 0.000,B 0.000,C 90.000,E1 58.456} C_DIS
LIN {X 0.054,Y -277.928,Z 738.306,A 0.000,B 0.000,C 90.000,E1 55.055} C_DIS
LIN {X -0.054,Y -270.707,Z 738.291,A 0.000,B 0.000,C 90.000,E1 52.316} C_DIS
LIN {X 0.065,Y -265.207,Z 738.279,A 0.000,B 0.000,C 90.000,E1 50.194} C_DIS
LIN {X 0.042,Y -259.598,Z 738.267,A 0.000,B 0.000,C 90.000,E1 48.081} C_DIS
LIN {X -0.104,Y -253.919,Z 738.255,A 0.000,B 0.000,C 90.000,E1 45.972} C_DIS
LIN {X -0.005,Y -248.201,Z 738.243,A 0.000,B 0.000,C 90.000,E1 43.785} C_DIS
LIN {X -0.019,Y -240.465,Z 738.227,A 0.000,B 0.000,C 90.000,E1 40.862} C_DIS
LIN {X -0.016,Y -232.787,Z 738.210,A 0.000,B 0.000,C 90.000,E1 37.890} C_DIS
LIN {X -0.118,Y -225.560,Z 738.194,A 0.000,B 0.000,C 90.000,E1 34.898} C_DIS
LIN {X -0.075,Y -217.223,Z 738.172,A 0.000,B 0.000,C 90.000,E1 31.052} C_DIS
LIN {X 0.066,Y -211.270,Z 738.155,A 0.000,B 0.000,C 90.000,E1 27.897} C_DIS
LIN {X -0.043,Y -206.110,Z 738.138,A 0.000,B 0.000,C 90.000,E1 24.771} C_DIS
LIN {X -0.073,Y -201.607,Z 738.120,A 0.000,B 0.000,C 90.000,E1 21.589} C_DIS
LIN {X 0.086,Y -197.110,Z 738.097,A 0.000,B 0.000,C 90.000,E1 17.511} C_DIS
LIN {X 0.006,Y -193.114,Z 738.070,A 0.000,B 0.000,C 90.000,E1 12.647} C_DIS
LIN {X 0.022,Y -190.323,Z 738.038,A 0.000,B 0.000,C 90.000,E1 6.891} C_DIS
LIN {X 0.033,Y -191.417,Z 737.965,A 0.000,B 0.000,C 90.000,E1 353.742} C_DIS
LIN {X 0.026,Y -194.543,Z 737.938,A 0.000,B 0.000,C 90.000,E1 348.814} C_DIS
LIN {X -0.048,Y -198.295,Z 737.915,A 0.000,B 0.000,C 90.000,E1 344.755} C_DIS
LIN {X 0.066,Y -202.945,Z 737.893,A 0.000,B 0.000,C 90.000,E1 340.678} C_DIS
LIN {X 0.103,Y -208.600,Z 737.871,A 0.000,B 0.000,C 90.000,E1 336.666} C_DIS
LIN {X -0.001,Y -215.155,Z 737.849,A 0.000,B 0.000,C 90.000,E1 332.743} C_DIS
LIN {X -0.086,Y -222.258,Z 737.827,A 0.000,B 0.000,C 90.000,E1 328.869} C_DIS
LIN {X -0.046,Y -230.035,Z 737.806,A 0.000,B 0.000,C 90.000,E1 325.022} C_DIS
LIN {X 0.007,Y -236.664,Z 737.789,A 0.000,B 0.000,C 90.000,E1 321.984} C_DIS
LIN {X 0.089,Y -245.695,Z 737.768,A 0.000,B 0.000,C 90.000,E1 318.243} C_DIS
LIN {X 0.072,Y -255.619,Z 737.748,A 0.000,B 0.000,C 90.000,E1 314.595} C_DIS
LIN {X -0.142,Y -266.602,Z 737.728,A 0.000,B 0.000,C 90.000,E1 311.067} C_DIS
LIN {X -0.020,Y -277.427,Z 737.710,A 0.000,B 0.000,C 90.000,E1 307.890} C_DIS
LIN {X 0.047,Y -290.678,Z 737.691,A 0.000,B 0.000,C 90.000,E1 304.452} C_DIS
LIN {X -0.040,Y -305.690,Z 737.673,A 0.000,B 0.000,C 90.000,E1 301.131} C_DIS
LIN {X 0.175,Y -319.081,Z 737.658,A 0.000,B 0.000,C 90.000,E1 298.487} C_DIS
LIN {X -0.037,Y -335.387,Z 737.643,A 0.000,B 0.000,C 90.000,E1 295.668} C_DIS
LIN {X -0.100,Y -351.054,Z 737.629,A 0.000,B 0.000,C 90.000,E1 293.206} C_DIS
LIN {X 0.106,Y -371.888,Z 737.612,A 0.000,B 0.000,C 90.000,E1 290.174} C_DIS
LIN {X -0.030,Y -392.639,Z 737.598,A 0.000,B 0.000,C 90.000,E1 287.583} C_DIS
LIN {X -0.101,Y -406.973,Z 737.588,A 0.000,B 0.000,C 90.000,E1 285.898} C_DIS
LIN {X -0.137,Y -421.122,Z 737.579,A 0.000,B 0.000,C 90.000,E1 284.245} C_DIS
LIN {X -0.096,Y -432.642,Z 737.571,A 0.000,B 0.000,C 90.000,E1 282.883} C_DIS
LIN {X -0.185,Y -441.530,Z 737.566,A 0.000,B 0.000,C 90.000,E1 281.827} C_DIS
LIN {X -0.017,Y -452.016,Z 737.558,A 0.000,B 0.000,C 90.000,E1 280.489} C_DIS
LIN {X 0.145,Y -464.110,Z 737.550,A 0.000,B 0.000,C 90.000,E1 278.916} C_DIS
LIN {X -0.187,Y -471.942,Z 737.544,A 0.000,B 0.000,C 90.000,E1 277.936} C_DIS
LIN {X -0.232,Y -477.284,Z 737.540,A 0.000,B 0.000,C 90.000,E1 277.182} C_DIS
LIN {X 0.249,Y -481.875,Z 737.536,A 0.000,B 0.000,C 90.000,E1 276.372} C_DIS
LIN {X -0.066,Y -484.540,Z 737.533,A 0.000,B 0.000,C 90.000,E1 275.910} C_DIS
LIN {X -0.055,Y -487.872,Z 737.529,A 0.000,B 0.000,C 90.000,E1 275.163} C_DIS
LIN {X 0.147,Y -489.586,Z 737.526,A 0.000,B 0.000,C 90.000,E1 274.645} C_DIS
LIN {X -0.170,Y -490.860,Z 737.523,A 0.000,B 0.000,C 90.000,E1 274.188} C_DIS
LIN {X 0.047,Y -491.771,Z 737.520,A 0.000,B 0.000,C 90.000,E1 273.669} C_DIS
LIN {X -0.249,Y -492.291,Z 737.518,A 0.000,B 0.000,C 90.000,E1 273.212} C_DIS
LIN {X -0.021,Y -492.398,Z 737.515,A 0.000,B 0.000,C 90.000,E1 272.694} C_DIS
LIN {X 0.184,Y -492.092,Z 737.512,A 0.000,B 0.000,C 90.000,E1 272.178} C_DIS
LIN {X -0.083,Y -491.395,Z 737.510,A 0.000,B 0.000,C 90.000,E1 271.718} C_DIS
LIN {X 0.123,Y -490.257,Z 737.507,A 0.000,B 0.000,C 90.000,E1 271.203} C_DIS
LIN {X -0.164,Y -488.651,Z 737.504,A 0.000,B 0.000,C 90.000,E1 270.745} C_DIS
LIN {X 0.032,Y -486.531,Z 737.501,A 0.000,B 0.000,C 90.000,E1 270.229} C_DIS
LIN {X 0.218,Y -483.847,Z 737.499,A 0.000,B 0.000,C 90.000,E1 269.714} C_DIS
LIN {X -0.099,Y -480.375,Z 737.496,A 0.000,B 0.000,C 90.000,E1 269.255} C_DIS
LIN {X 0.048,Y -476.024,Z 737.493,A 0.000,B 0.000,C 90.000,E1 268.740} C_DIS
LIN {X -0.128,Y -473.447,Z 737.492,A 0.000,B 0.000,C 90.000,E1 268.511} C_DIS
LIN {X 0.211,Y -467.649,Z 737.489,A 0.000,B 0.000,C 90.000,E1 267.993} C_DIS
LIN {X -0.225,Y -464.427,Z 737.488,A 0.000,B 0.000,C 90.000,E1 267.822} C_DIS
LIN {X -0.129,Y -457.826,Z 737.486,A 0.000,B 0.000,C 90.000,E1 267.421} C_DIS
LIN {X -0.070,Y -454.528,Z 737.485,A 0.000,B 0.000,C 90.000,E1 267.249} C_DIS
LIN {X -0.121,Y -447.264,Z 737.483,A 0.000,B 0.000,C 90.000,E1 266.963} C_DIS
LIN {X -0.065,Y -439.587,Z 737.482,A 0.000,B 0.000,C 90.000,E1 266.731} C_DIS
LIN {X -0.015,Y -431.321,Z 737.481,A 0.000,B 0.000,C 90.000,E1 266.560} C_DIS
LIN {X 0.165,Y -422.793,Z 737.480,A 0.000,B 0.000,C 90.000,E1 266.445} C_DIS
LIN {X 0.085,Y -421.097,Z 737.480,A 0.000,B 0.000,C 90.000,E1 266.445} C_DIS
LIN {X 0.002,Y -180.944,Z 737.480,A 0.000,B 0.000,C 90.000,E1 266.445} C_DIS
LIN {X -0.020,Y -180.774,Z 737.471,A 0.000,B 0.000,C 90.000,E1 264.723} C_DIS
LIN {X 0.052,Y -178.869,Z 737.443,A 0.000,B 0.000,C 90.000,E1 259.634} C_DIS
LIN {X -0.048,Y -175.912,Z 737.414,A 0.000,B 0.000,C 90.000,E1 254.574} C_DIS
LIN {X 0.008,Y -174.602,Z 737.405,A 0.000,B 0.000,C 90.000,E1 252.851} C_DIS
LIN {X -0.065,Y -171.584,Z 737.381,A 0.000,B 0.000,C 90.000,E1 248.592} C_DIS
LIN {X -0.075,Y -167.806,Z 737.357,A 0.000,B 0.000,C 90.000,E1 244.280} C_DIS
LIN {X -0.057,Y -166.527,Z 737.347,A 0.000,B 0.000,C 90.000,E1 242.538} C_DIS
LIN {X 0.077,Y -162.526,Z 737.323,A 0.000,B 0.000,C 90.000,E1 238.122} C_DIS
LIN {X 0.049,Y -161.200,Z 737.313,A 0.000,B 0.000,C 90.000,E1 236.373} C_DIS
LIN {X -0.050,Y -157.210,Z 737.289,A 0.000,B 0.000,C 90.000,E1 231.984} C_DIS
LIN {X -0.026,Y -155.938,Z 737.279,A 0.000,B 0.000,C 90.000,E1 230.194} C_DIS
LIN {X -0.066,Y -152.189,Z 737.254,A 0.000,B 0.000,C 90.000,E1 225.729} C_DIS
LIN {X -0.044,Y -150.436,Z 737.239,A 0.000,B 0.000,C 90.000,E1 223.014} C_DIS
LIN {X -0.017,Y -147.163,Z 737.214,A 0.000,B 0.000,C 90.000,E1 218.463} C_DIS
LIN {X -0.050,Y -145.178,Z 737.193,A 0.000,B 0.000,C 90.000,E1 214.818} C_DIS
LIN {X -0.015,Y -142.325,Z 737.163,A 0.000,B 0.000,C 90.000,E1 209.283} C_DIS
LIN {X -0.020,Y -141.715,Z 737.152,A 0.000,B 0.000,C 90.000,E1 207.436} C_DIS
LIN {X 0.028,Y -139.474,Z 737.116,A 0.000,B 0.000,C 90.000,E1 200.918} C_DIS
LIN {X 0.018,Y -138.970,Z 737.101,A 0.000,B 0.000,C 90.000,E1 198.127} C_DIS
LIN {X 0.008,Y -138.330,Z 737.054,A 0.000,B 0.000,C 90.000,E1 189.726} C_DIS
LIN {X 0.011,Y -139.437,Z 737.007,A 0.000,B 0.000,C 90.000,E1 181.318} C_DIS
LIN {X -0.050,Y -140.968,Z 736.976,A 0.000,B 0.000,C 90.000,E1 175.755} C_DIS
LIN {X 0.042,Y -142.724,Z 736.956,A 0.000,B 0.000,C 90.000,E1 172.008} C_DIS
LIN {X -0.001,Y -145.107,Z 736.930,A 0.000,B 0.000,C 90.000,E1 167.409} C_DIS
LIN {X -0.006,Y -147.731,Z 736.910,A 0.000,B 0.000,C 90.000,E1 163.740} C_DIS
LIN {X 0.076,Y -150.393,Z 736.889,A 0.000,B 0.000,C 90.000,E1 160.061} C_DIS
LIN {X -0.049,Y -153.827,Z 736.869,A 0.000,B 0.000,C 90.000,E1 156.485} C_DIS
LIN {X 0.010,Y -157.238,Z 736.849,A 0.000,B 0.000,C 90.000,E1 152.871} C_DIS
LIN {X -0.049,Y -161.408,Z 736.830,A 0.000,B 0.000,C 90.000,E1 149.331} C_DIS
LIN {X -0.039,Y -165.610,Z 736.810,A 0.000,B 0.000,C 90.000,E1 145.801} C_DIS
LIN {X 0.080,Y -170.536,Z 736.791,A 0.000,B 0.000,C 90.000,E1 142.271} C_DIS
LIN {X -0.011,Y -175.415,Z 736.771,A 0.000,B 0.000,C 90.000,E1 138.852} C_DIS
LIN {X -0.021,Y -181.039,Z 736.752,A 0.000,B 0.000,C 90.000,E1 135.445} C_DIS
LIN {X -0.027,Y -186.473,Z 736.734,A 0.000,B 0.000,C 90.000,E1 132.081} C_DIS
LIN {X 0.070,Y -191.545,Z 736.718,A 0.000,B 0.000,C 90.000,E1 129.277} C_DIS
LIN {X 0.091,Y -191.800,Z 736.717,A 0.000,B 0.000,C 90.000,E1 129.116} C_DIS
LIN {X 0.104,Y -290.586,Z 736.717,A 0.000,B 0.000,C 90.000,E1 129.116} C_DIS
LIN {X 0.000,Y -292.033,Z 736.717,A 0.000,B 0.000,C 90.000,E1 129.116} C_DIS
LIN {X 0.116,Y -296.341,Z 736.716,A 0.000,B 0.000,C 90.000,E1 128.910} C_DIS
LIN {X 0.000,Y -298.681,Z 736.715,A 0.000,B 0.000,C 90.000,E1 128.749} C_DIS
LIN {X -0.090,Y -302.537,Z 736.713,A 0.000,B 0.000,C 90.000,E1 128.302} C_DIS
LIN {X -0.059,Y -304.408,Z 736.711,A 0.000,B 0.000,C 90.000,E1 127.971} C_DIS
LIN {X -0.082,Y -305.871,Z 736.709,A 0.000,B 0.000,C 90.000,E1 127.649} C_DIS
LIN {X 0.145,Y -307.971,Z 736.705,A 0.000,B 0.000,C 90.000,E1 126.950} C_DIS
LIN {X 0.124,Y -317.814,Z 736.687,A 0.000,B 0.000,C 90.000,E1 123.706} C_DIS
LIN {X -0.102,Y -327.973,Z 736.671,A 0.000,B 0.000,C 90.000,E1 120.875} C_DIS
LIN {X 0.072,Y -339.470,Z 736.656,A 0.000,B 0.000,C 90.000,E1 118.025} C_DIS
LIN {X -0.056,Y -352.402,Z 736.640,A 0.000,B 0.000,C 90.000,E1 115.283} C_DIS
LIN {X -0.185,Y -365.198,Z 736.627,A 0.000,B 0.000,C 90.000,E1 112.898} C_DIS
LIN {X 0.207,Y -379.312,Z 736.614,A 0.000,B 0.000,C 90.000,E1 110.482} C_DIS
LIN {X -0.164,Y -394.846,Z 736.601,A 0.000,B 0.000,C 90.000,E1 108.236} C_DIS
LIN {X -0.020,Y -411.912,Z 736.589,A 0.000,B 0.000,C 90.000,E1 105.969} C_DIS
LIN {X 0.053,Y -430.635,Z 736.577,A 0.000,B 0.000,C 90.000,E1 103.772} C_DIS
LIN {X -0.074,Y -450.617,Z 736.565,A 0.000,B 0.000,C 90.000,E1 101.715} C_DIS
LIN {X 0.098,Y -468.504,Z 736.556,A 0.000,B 0.000,C 90.000,E1 100.018} C_DIS
LIN {X 0.016,Y -470.492,Z 736.554,A 0.000,B 0.000,C 90.000,E1 99.792} C_DIS
LIN {X 0.013,Y -472.004,Z 736.553,A 0.000,B 0.000,C 90.000,E1 99.557} C_DIS
LIN {X -0.132,Y -473.235,Z 736.552,A 0.000,B 0.000,C 90.000,E1 99.321} C_DIS
LIN {X 0.189,Y -474.136,Z 736.550,A 0.000,B 0.000,C 90.000,E1 99.029} C_DIS
LIN {X -0.162,Y -475.108,Z 736.547,A 0.000,B 0.000,C 90.000,E1 98.568} C_DIS
LIN {X -0.038,Y -475.098,Z 736.545,A 0.000,B 0.000,C 90.000,E1 98.049} C_DIS
LIN {X 0.095,Y -474.109,Z 736.542,A 0.000,B 0.000,C 90.000,E1 97.530} C_DIS
LIN {X -0.241,Y -471.972,Z 736.539,A 0.000,B 0.000,C 90.000,E1 97.068} C_DIS
LIN {X -0.043,Y -454.139,Z 736.524,A 0.000,B 0.000,C 90.000,E1 94.245} C_DIS
LIN {X -0.206,Y -439.282,Z 736.509,A 0.000,B 0.000,C 90.000,E1 91.661} C_DIS
LIN {X 0.185,Y -431.750,Z 736.502,A 0.000,B 0.000,C 90.000,E1 90.286} C_DIS
LIN {X -0.148,Y -420.823,Z 736.491,A 0.000,B 0.000,C 90.000,E1 88.453} C_DIS
LIN {X 0.082,Y -411.387,Z 736.482,A 0.000,B 0.000,C 90.000,E1 86.788} C_DIS
LIN {X 0.197,Y -400.253,Z 736.471,A 0.000,B 0.000,C 90.000,E1 84.837} C_DIS
LIN {X 0.146,Y -387.541,Z 736.459,A 0.000,B 0.000,C 90.000,E1 82.591} C_DIS
LIN {X -0.089,Y -373.685,Z 736.445,A 0.000,B 0.000,C 90.000,E1 80.038} C_DIS
LIN {X -0.175,Y -360.345,Z 736.430,A 0.000,B 0.000,C 90.000,E1 77.409} C_DIS
LIN {X -0.049,Y -348.952,Z 736.417,A 0.000,B 0.000,C 90.000,E1 74.991} C_DIS
LIN {X -0.031,Y -336.338,Z 736.401,A 0.000,B 0.000,C 90.000,E1 72.236} C_DIS
LIN {X 0.124,Y -322.954,Z 736.384,A 0.000,B 0.000,C 90.000,E1 69.082} C_DIS
LIN {X -0.084,Y -310.681,Z 736.366,A 0.000,B 0.000,C 90.000,E1 65.921} C_DIS
LIN {X 0.033,Y -298.815,Z 736.346,A 0.000,B 0.000,C 90.000,E1 62.308} C_DIS
LIN {X -0.052,Y -288.941,Z 736.328,A 0.000,B 0.000,C 90.000,E1 58.997} C_DIS
LIN {X 0.019,Y -279.623,Z 736.309,A 0.000,B 0.000,C 90.000,E1 55.595} C_DIS
LIN {X 0.011,Y -272.435,Z 736.294,A 0.000,B 0.000,C 90.000,E1 52.844} C_DIS
LIN {X 0.159,Y -267.002,Z 736.282,A 0.000,B 0.000,C 90.000,E1 50.723} C_DIS
LIN {X -0.005,Y -261.422,Z 736.270,A 0.000,B 0.000,C 90.000,E1 48.647} C_DIS
LIN {X -0.066,Y -253.885,Z 736.254,A 0.000,B 0.000,C 90.000,E1 45.810} C_DIS
LIN {X 0.032,Y -248.140,Z 736.242,A 0.000,B 0.000,C 90.000,E1 43.623} C_DIS
LIN {X 0.013,Y -240.382,Z 736.226,A 0.000,B 0.000,C 90.000,E1 40.701} C_DIS
LIN {X -0.058,Y -230.830,Z 736.205,A 0.000,B 0.000,C 90.000,E1 36.996} C_DIS
LIN {X 0.152,Y -223.748,Z 736.189,A 0.000,B 0.000,C 90.000,E1 33.913} C_DIS
LIN {X 0.005,Y -217.144,Z 736.172,A 0.000,B 0.000,C 90.000,E1 30.875} C_DIS
LIN {X -0.037,Y -211.195,Z 736.154,A 0.000,B 0.000,C 90.000,E1 27.769} C_DIS
LIN {X -0.055,Y -204.849,Z 736.132,A 0.000,B 0.000,C 90.000,E1 23.823} C_DIS
LIN {X -0.006,Y -200.566,Z 736.115,A 0.000,B 0.000,C 90.000,E1 20.610} C_DIS
LIN {X 0.000,Y -196.338,Z 736.092,A 0.000,B 0.000,C 90.000,E1 16.567} C_DIS
LIN {X 0.046,Y -192.614,Z 736.065,A 0.000,B 0.000,C 90.000,E1 11.658} C_DIS
LIN {X -0.051,Y -189.960,Z 736.028,A 0.000,B 0.000,C 90.000,E1 5.106} C_DIS
LIN {X 0.086,Y -191.156,Z 735.970,A 0.000,B 0.000,C 90.000,E1 354.552} C_DIS
LIN {X 0.031,Y -193.997,Z 735.942,A 0.000,B 0.000,C 90.000,E1 349.634} C_DIS
LIN {X -0.059,Y -197.574,Z 735.920,A 0.000,B 0.000,C 90.000,E1 345.574} C_DIS
LIN {X -0.017,Y -202.052,Z 735.897,A 0.000,B 0.000,C 90.000,E1 341.511} C_DIS
LIN {X 0.035,Y -207.507,Z 735.875,A 0.000,B 0.000,C 90.000,E1 337.486} C_DIS
LIN {X 0.085,Y -213.900,Z 735.853,A 0.000,B 0.000,C 90.000,E1 333.512} C_DIS
LIN {X 0.049,Y -220.877,Z 735.831,A 0.000,B 0.000,C 90.000,E1 329.616} C_DIS
LIN {X -0.084,Y -228.477,Z 735.810,A 0.000,B 0.000,C 90.000,E1 325.801} C_DIS
LIN {X 0.040,Y -236.713,Z 735.789,A 0.000,B 0.000,C 90.000,E1 321.984} C_DIS
LIN {X 0.124,Y -245.726,Z 735.768,A 0.000,B 0.000,C 90.000,E1 318.243} C_DIS
LIN {X 0.109,Y -255.614,Z 735.748,A 0.000,B 0.000,C 90.000,E1 314.595} C_DIS
LIN {X 0.040,Y -265.481,Z 735.730,A 0.000,B 0.000,C 90.000,E1 311.391} C_DIS
LIN {X -0.078,Y -276.159,Z 735.712,A 0.000,B 0.000,C 90.000,E1 308.257} C_DIS
LIN {X -0.050,Y -289.311,Z 735.693,A 0.000,B 0.000,C 90.000,E1 304.818} C_DIS
LIN {X -0.019,Y -304.133,Z 735.675,A 0.000,B 0.000,C 90.000,E1 301.465} C_DIS
LIN {X 0.098,Y -315.608,Z 735.662,A 0.000,B 0.000,C 90.000,E1 299.155} C_DIS
LIN {X 0.086,Y -331.685,Z 735.646,A 0.000,B 0.000,C 90.000,E1 296.283} C_DIS
LIN {X -0.077,Y -345.084,Z 735.634,A 0.000,B 0.000,C 90.000,E1 294.131} C_DIS
LIN {X -0.134,Y -363.239,Z 735.619,A 0.000,B 0.000,C 90.000,E1 291.408} C_DIS
LIN {X -0.130,Y -376.237,Z 735.609,A 0.000,B 0.000,C 90.000,E1 289.631} C_DIS
LIN {X 0.024,Y -392.487,Z 735.598,A 0.000,B 0.000,C 90.000,E1 287.583} C_DIS
LIN {X -0.046,Y -406.783,Z 735.588,A 0.000,B 0.000,C 90.000,E1 285.898} C_DIS
LIN {X -0.085,Y -420.925,Z 735.579,A 0.000,B 0.000,C 90.000,E1 284.245} C_DIS
LIN {X -0.045,Y -432.434,Z 735.572,A 0.000,B 0.000,C 90.000,E1 282.883} C_DIS
LIN {X -0.137,Y -441.311,Z 735.566,A 0.000,B 0.000,C 90.000,E1 281.827} C_DIS
LIN {X 0.030,Y -451.801,Z 735.558,A 0.000,B 0.000,C 90.000,E1 280.489} C_DIS
LIN {X 0.188,Y -463.903,Z 735.550,A 0.000,B 0.000,C 90.000,E1 278.916} C_DIS
LIN {X -0.144,Y -471.745,Z 735.544,A 0.000,B 0.000,C 90.000,E1 277.936} C_DIS
LIN {X -0.191,Y -477.095,Z 735.540,A 0.000,B 0.000,C 90.000,E1 277.182} C_DIS
LIN {X -0.190,Y -481.688,Z 735.536,A 0.000,B 0.000,C 90.000,E1 276.429} C_DIS
LIN {X -0.027,Y -484.352,Z 735.533,A 0.000,B 0.000,C 90.000,E1 275.910} C_DIS
LIN {X 0.154,Y -486.655,Z 735.530,A 0.000,B 0.000,C 90.000,E1 275.391} C_DIS
LIN {X 0.185,Y -489.385,Z 735.526,A 0.000,B 0.000,C 90.000,E1 274.645} C_DIS
LIN {X -0.135,Y -490.663,Z 735.523,A 0.000,B 0.000,C 90.000,E1 274.188} C_DIS
LIN {X 0.082,Y -491.571,Z 735.520,A 0.000,B 0.000,C 90.000,E1 273.669} C_DIS
LIN {X -0.215,Y -492.014,Z 735.518,A 0.000,B 0.000,C 90.000,E1 273.212} C_DIS
LIN {X 0.011,Y -492.153,Z 735.515,A 0.000,B 0.000,C 90.000,E1 272.694} C_DIS
LIN {X 0.215,Y -491.865,Z 735.512,A 0.000,B 0.000,C 90.000,E1 272.178} C_DIS
LIN {X -0.053,Y -491.142,Z 735.510,A 0.000,B 0.000,C 90.000,E1 271.718} C_DIS
LIN {X 0.151,Y -490.027,Z 735.507,A 0.000,B 0.000,C 90.000,E1 271.203} C_DIS
LIN {X -0.137,Y -488.433,Z 735.504,A 0.000,B 0.000,C 90.000,E1 270.745} C_DIS
LIN {X 0.058,Y -486.358,Z 735.501,A 0.000,B 0.000,C 90.000,E1 270.229} C_DIS
LIN {X -0.242,Y -483.706,Z 735.499,A 0.000,B 0.000,C 90.000,E1 269.771} C_DIS
LIN {X -0.075,Y -480.270,Z 735.496,A 0.000,B 0.000,C 90.000,E1 269.255} C_DIS
LIN {X 0.071,Y -476.003,Z 735.493,A 0.000,B 0.000,C 90.000,E1 268.740} C_DIS
LIN {X -0.106,Y -473.448,Z 735.492,A 0.000,B 0.000,C 90.000,E1 268.511} C_DIS
LIN {X 0.227,Y -467.708,Z 735.489,A 0.000,B 0.000,C 90.000,E1 267.993} C_DIS
LIN {X 0.049,Y -461.419,Z 735.487,A 0.000,B 0.000,C 90.000,E1 267.593} C_DIS
LIN {X -0.093,Y -454.629,Z 735.485,A 0.000,B 0.000,C 90.000,E1 267.249} C_DIS
LIN {X -0.155,Y -447.308,Z 735.483,A 0.000,B 0.000,C 90.000,E1 266.963} C_DIS
LIN {X -0.142,Y -439.509,Z 735.482,A 0.000,B 0.000,C 90.000,E1 266.731} C_DIS
LIN {X -0.125,Y -430.986,Z 735.481,A 0.000,B 0.000,C 90.000,E1 266.560} C_DIS
LIN {X 0.058,Y -422.346,Z 735.480,A 0.000,B 0.000,C 90.000,E1 266.445} C_DIS
LIN {X -0.022,Y -420.177,Z 735.480,A 0.000,B 0.000,C 90.000,E1 266.445} C_DIS
LIN {X -0.044,Y -180.944,Z 735.480,A 0.000,B 0.000,C 90.000,E1 266.445} C_DIS
LIN {X -0.064,Y -180.768,Z 735.471,A 0.000,B 0.000,C 90.000,E1 264.723} C_DIS
LIN {X 0.008,Y -178.863,Z 735.442,A 0.000,B 0.000,C 90.000,E1 259.634} C_DIS
LIN {X -0.091,Y -175.906,Z 735.414,A 0.000,B 0.000,C 90.000,E1 254.574} C_DIS
LIN {X 0.017,Y -174.590,Z 735.405,A 0.000,B 0.000,C 90.000,E1 252.834} C_DIS
LIN {X 0.052,Y -171.573,Z 735.381,A 0.000,B 0.000,C 90.000,E1 248.539} C_DIS
LIN {X 0.034,Y -167.795,Z 735.357,A 0.000,B 0.000,C 90.000,E1 244.229} C_DIS
LIN {X 0.048,Y -166.512,Z 735.347,A 0.000,B 0.000,C 90.000,E1 242.487} C_DIS
LIN {X 0.043,Y -163.220,Z 735.328,A 0.000,B 0.000,C 90.000,E1 238.997} C_DIS
LIN {X 0.008,Y -161.187,Z 735.313,A 0.000,B 0.000,C 90.000,E1 236.373} C_DIS
LIN {X 0.007,Y -157.198,Z 735.289,A 0.000,B 0.000,C 90.000,E1 231.949} C_DIS
LIN {X 0.053,Y -155.927,Z 735.279,A 0.000,B 0.000,C 90.000,E1 230.150} C_DIS
LIN {X 0.003,Y -152.178,Z 735.254,A 0.000,B 0.000,C 90.000,E1 225.688} C_DIS
LIN {X 0.018,Y -150.426,Z 735.239,A 0.000,B 0.000,C 90.000,E1 222.975} C_DIS
LIN {X -0.056,Y -147.154,Z 735.214,A 0.000,B 0.000,C 90.000,E1 218.463} C_DIS
LIN {X 0.031,Y -145.168,Z 735.193,A 0.000,B 0.000,C 90.000,E1 214.771} C_DIS
LIN {X -0.053,Y -142.319,Z 735.163,A 0.000,B 0.000,C 90.000,E1 209.283} C_DIS
LIN {X 0.067,Y -141.708,Z 735.152,A 0.000,B 0.000,C 90.000,E1 207.385} C_DIS
LIN {X -0.010,Y -139.471,Z 735.116,A 0.000,B 0.000,C 90.000,E1 200.918} C_DIS
LIN {X 0.044,Y -139.202,Z 735.106,A 0.000,B 0.000,C 90.000,E1 199.033} C_DIS
LIN {X -0.029,Y -138.328,Z 735.054,A 0.000,B 0.000,C 90.000,E1 189.726} C_DIS
LIN {X -0.027,Y -139.440,Z 735.007,A 0.000,B 0.000,C 90.000,E1 181.318} C_DIS
LIN {X 0.053,Y -140.974,Z 734.976,A 0.000,B 0.000,C 90.000,E1 175.698} C_DIS
LIN {X 0.003,Y -142.730,Z 734.956,A 0.000,B 0.000,C 90.000,E1 172.008} C_DIS
LIN {X -0.039,Y -145.116,Z 734.930,A 0.000,B 0.000,C 90.000,E1 167.409} C_DIS
LIN {X -0.046,Y -147.740,Z 734.910,A 0.000,B 0.000,C 90.000,E1 163.740} C_DIS
LIN {X 0.037,Y -150.405,Z 734.889,A 0.000,B 0.000,C 90.000,E1 160.061} C_DIS
LIN {X 0.052,Y -153.843,Z 734.869,A 0.000,B 0.000,C 90.000,E1 156.433} C_DIS
LIN {X -0.030,Y -157.253,Z 734.849,A 0.000,B 0.000,C 90.000,E1 152.871} C_DIS
LIN {X 0.047,Y -161.428,Z 734.829,A 0.000,B 0.000,C 90.000,E1 149.282} C_DIS
LIN {X -0.082,Y -165.628,Z 734.810,A 0.000,B 0.000,C 90.000,E1 145.801} C_DIS
LIN {X 0.038,Y -170.559,Z 734.790,A 0.000,B 0.000,C 90.000,E1 142.271} C_DIS
LIN {X -0.054,Y -175.437,Z 734.771,A 0.000,B 0.000,C 90.000,E1 138.852} C_DIS
LIN {X 0.062,Y -181.060,Z 734.752,A 0.000,B 0.000,C 90.000,E1 135.405} C_DIS
LIN {X -0.072,Y -186.497,Z 734.734,A 0.000,B 0.000,C 90.000,E1 132.081} C_DIS
LIN {X 0.026,Y -191.567,Z 734.718,A 0.000,B 0.000,C 90.000,E1 129.277} C_DIS
LIN {X 0.017,Y -191.776,Z 734.718,A 0.000,B 0.000,C 90.000,E1 129.152} C_DIS
LIN {X -0.008,Y -290.791,Z 734.718,A 0.000,B 0.000,C 90.000,E1 129.152} C_DIS
LIN {X -0.067,Y -293.073,Z 734.717,A 0.000,B 0.000,C 90.000,E1 129.116} C_DIS
LIN {X 0.047,Y -296.717,Z 734.716,A 0.000,B 0.000,C 90.000,E1 128.910} C_DIS
LIN {X -0.071,Y -298.936,Z 734.715,A 0.000,B 0.000,C 90.000,E1 128.749} C_DIS
LIN {X -0.042,Y -302.808,Z 734.713,A 0.000,B 0.000,C 90.000,E1 128.257} C_DIS
LIN {X -0.094,Y -304.631,Z 734.711,A 0.000,B 0.000,C 90.000,E1 127.935} C_DIS
LIN {X -0.094,Y -306.055,Z 734.709,A 0.000,B 0.000,C 90.000,E1 127.604} C_DIS
LIN {X -0.109,Y -308.082,Z 734.705,A 0.000,B 0.000,C 90.000,E1 126.950} C_DIS
LIN {X -0.133,Y -317.946,Z 734.687,A 0.000,B 0.000,C 90.000,E1 123.706} C_DIS
LIN {X 0.086,Y -328.126,Z 734.671,A 0.000,B 0.000,C 90.000,E1 120.797} C_DIS
LIN {X 0.105,Y -339.645,Z 734.656,A 0.000,B 0.000,C 90.000,E1 117.975} C_DIS
LIN {X 0.141,Y -352.601,Z 734.640,A 0.000,B 0.000,C 90.000,E1 115.207} C_DIS
LIN {X 0.017,Y -365.420,Z 734.627,A 0.000,B 0.000,C 90.000,E1 112.823} C_DIS
LIN {X -0.075,Y -379.558,Z 734.614,A 0.000,B 0.000,C 90.000,E1 110.482} C_DIS
LIN {X -0.076,Y -395.119,Z 734.601,A 0.000,B 0.000,C 90.000,E1 108.181} C_DIS
LIN {X 0.196,Y -412.214,Z 734.589,A 0.000,B 0.000,C 90.000,E1 105.898} C_DIS
LIN {X -0.246,Y -430.969,Z 734.576,A 0.000,B 0.000,C 90.000,E1 103.772} C_DIS
LIN {X 0.078,Y -450.964,Z 734.565,A 0.000,B 0.000,C 90.000,E1 101.658} C_DIS
LIN {X -0.182,Y -468.807,Z 734.556,A 0.000,B 0.000,C 90.000,E1 100.018} C_DIS
LIN {X 0.254,Y -470.744,Z 734.554,A 0.000,B 0.000,C 90.000,E1 99.726} C_DIS
LIN {X 0.150,Y -472.217,Z 734.553,A 0.000,B 0.000,C 90.000,E1 99.500} C_DIS
LIN {X 0.006,Y -473.395,Z 734.551,A 0.000,B 0.000,C 90.000,E1 99.265} C_DIS
LIN {X -0.140,Y -474.254,Z 734.550,A 0.000,B 0.000,C 90.000,E1 99.029} C_DIS
LIN {X -0.021,Y -475.153,Z 734.547,A 0.000,B 0.000,C 90.000,E1 98.511} C_DIS
LIN {X 0.104,Y -475.076,Z 734.544,A 0.000,B 0.000,C 90.000,E1 97.992} C_DIS
LIN {X -0.232,Y -474.014,Z 734.542,A 0.000,B 0.000,C 90.000,E1 97.530} C_DIS
LIN {X 0.100,Y -473.066,Z 734.540,A 0.000,B 0.000,C 90.000,E1 97.239} C_DIS
LIN {X -0.040,Y -471.783,Z 734.539,A 0.000,B 0.000,C 90.000,E1 97.004} C_DIS
LIN {X -0.114,Y -452.380,Z 734.522,A 0.000,B 0.000,C 90.000,E1 93.955} C_DIS
LIN {X -0.087,Y -439.079,Z 734.509,A 0.000,B 0.000,C 90.000,E1 91.604} C_DIS
LIN {X 0.017,Y -429.992,Z 734.500,A 0.000,B 0.000,C 90.000,E1 90.000} C_DIS
LIN {X 0.088,Y -419.092,Z 734.490,A 0.000,B 0.000,C 90.000,E1 88.108} C_DIS
LIN {X -0.069,Y -408.052,Z 734.479,A 0.000,B 0.000,C 90.000,E1 86.216} C_DIS
LIN {X 0.008,Y -396.883,Z 734.468,A 0.000,B 0.000,C 90.000,E1 84.261} C_DIS
LIN {X -0.064,Y -384.279,Z 734.456,A 0.000,B 0.000,C 90.000,E1 82.008} C_DIS
LIN {X -0.004,Y -372.034,Z 734.443,A 0.000,B 0.000,C 90.000,E1 79.690} C_DIS
LIN {X -0.108,Y -360.253,Z 734.430,A 0.000,B 0.000,C 90.000,E1 77.353} C_DIS
LIN {X 0.010,Y -348.862,Z 734.416,A 0.000,B 0.000,C 90.000,E1 74.936} C_DIS
LIN {X 0.019,Y -336.278,Z 734.401,A 0.000,B 0.000,C 90.000,E1 72.181} C_DIS
LIN {X -0.136,Y -322.923,Z 734.384,A 0.000,B 0.000,C 90.000,E1 69.082} C_DIS
LIN {X -0.051,Y -310.702,Z 734.366,A 0.000,B 0.000,C 90.000,E1 65.869} C_DIS
LIN {X -0.069,Y -298.905,Z 734.346,A 0.000,B 0.000,C 90.000,E1 62.281} C_DIS
LIN {X -0.034,Y -289.069,Z 734.327,A 0.000,B 0.000,C 90.000,E1 58.948} C_DIS
LIN {X 0.031,Y -279.807,Z 734.309,A 0.000,B 0.000,C 90.000,E1 55.548} C_DIS
LIN {X -0.014,Y -274.449,Z 734.297,A 0.000,B 0.000,C 90.000,E1 53.497} C_DIS
LIN {X 0.004,Y -269.073,Z 734.286,A 0.000,B 0.000,C 90.000,E1 51.412} C_DIS
LIN {X 0.049,Y -263.542,Z 734.274,A 0.000,B 0.000,C 90.000,E1 49.299} C_DIS
LIN {X 0.057,Y -256.030,Z 734.258,A 0.000,B 0.000,C 90.000,E1 46.458} C_DIS
LIN {X 0.014,Y -250.319,Z 734.246,A 0.000,B 0.000,C 90.000,E1 44.312} C_DIS
LIN {X 0.045,Y -244.499,Z 734.234,A 0.000,B 0.000,C 90.000,E1 42.123} C_DIS
LIN {X -0.011,Y -238.643,Z 734.222,A 0.000,B 0.000,C 90.000,E1 39.930} C_DIS
LIN {X 0.086,Y -229.195,Z 734.201,A 0.000,B 0.000,C 90.000,E1 36.171} C_DIS
LIN {X -0.130,Y -220.524,Z 734.180,A 0.000,B 0.000,C 90.000,E1 32.418} C_DIS
LIN {X 0.024,Y -214.241,Z 734.163,A 0.000,B 0.000,C 90.000,E1 29.283} C_DIS
LIN {X -0.009,Y -208.673,Z 734.145,A 0.000,B 0.000,C 90.000,E1 26.155} C_DIS
LIN {X -0.089,Y -202.718,Z 734.123,A 0.000,B 0.000,C 90.000,E1 22.206} C_DIS
LIN {X -0.080,Y -198.018,Z 734.101,A 0.000,B 0.000,C 90.000,E1 18.181} C_DIS
LIN {X -0.081,Y -194.371,Z 734.078,A 0.000,B 0.000,C 90.000,E1 14.120} C_DIS
LIN {X -0.089,Y -191.434,Z 734.051,A 0.000,B 0.000,C 90.000,E1 9.208} C_DIS
LIN {X -0.032,Y -190.917,Z 733.974,A 0.000,B 0.000,C 90.000,E1 355.412} C_DIS
LIN {X 0.073,Y -193.512,Z 733.947,A 0.000,B 0.000,C 90.000,E1 350.443} C_DIS
LIN {X 0.077,Y -196.884,Z 733.924,A 0.000,B 0.000,C 90.000,E1 346.353} C_DIS
LIN {X 0.032,Y -201.200,Z 733.902,A 0.000,B 0.000,C 90.000,E1 342.308} C_DIS
LIN {X 0.055,Y -206.429,Z 733.879,A 0.000,B 0.000,C 90.000,E1 338.284} C_DIS
LIN {X -0.014,Y -212.683,Z 733.857,A 0.000,B 0.000,C 90.000,E1 334.332} C_DIS
LIN {X 0.002,Y -219.522,Z 733.836,A 0.000,B 0.000,C 90.000,E1 330.411} C_DIS
LIN {X 0.016,Y -226.952,Z 733.814,A 0.000,B 0.000,C 90.000,E1 326.548} C_DIS
LIN {X 0.049,Y -233.405,Z 733.797,A 0.000,B 0.000,C 90.000,E1 323.497} C_DIS
LIN {X 0.059,Y -242.040,Z 733.776,A 0.000,B 0.000,C 90.000,E1 319.747} C_DIS
LIN {X 0.113,Y -251.554,Z 733.756,A 0.000,B 0.000,C 90.000,E1 316.053} C_DIS
LIN {X -0.094,Y -261.046,Z 733.738,A 0.000,B 0.000,C 90.000,E1 312.852} C_DIS
LIN {X 0.005,Y -271.300,Z 733.720,A 0.000,B 0.000,C 90.000,E1 309.644} C_DIS
LIN {X 0.047,Y -283.942,Z 733.701,A 0.000,B 0.000,C 90.000,E1 306.171} C_DIS
LIN {X 0.083,Y -295.053,Z 733.686,A 0.000,B 0.000,C 90.000,E1 303.452} C_DIS
LIN {X 0.151,Y -310.558,Z 733.668,A 0.000,B 0.000,C 90.000,E1 300.129} C_DIS
LIN {X -0.061,Y -328.033,Z 733.650,A 0.000,B 0.000,C 90.000,E1 296.950} C_DIS
LIN {X -0.155,Y -341.119,Z 733.637,A 0.000,B 0.000,C 90.000,E1 294.771} C_DIS
LIN {X 0.064,Y -354.990,Z 733.626,A 0.000,B 0.000,C 90.000,E1 292.589} C_DIS
LIN {X -0.168,Y -373.853,Z 733.611,A 0.000,B 0.000,C 90.000,E1 289.939} C_DIS
LIN {X 0.148,Y -392.259,Z 733.598,A 0.000,B 0.000,C 90.000,E1 287.583} C_DIS
LIN {X 0.078,Y -406.527,Z 733.588,A 0.000,B 0.000,C 90.000,E1 285.898} C_DIS
LIN {X 0.039,Y -420.641,Z 733.579,A 0.000,B 0.000,C 90.000,E1 284.245} C_DIS
LIN {X 0.083,Y -432.150,Z 733.572,A 0.000,B 0.000,C 90.000,E1 282.883} C_DIS
LIN {X 0.203,Y -443.159,Z 733.564,A 0.000,B 0.000,C 90.000,E1 281.535} C_DIS
